      E_STATION_CTRL.STATION_ENABLE:
        IF (_wEnable = _wEnableProcess)
        THEN
          InitSerialTargets();
          _eProcessState            := E_STATION_STATE.STATION_DETECT_MOVER;
        END_IF
    END_CASE
END_CASE
//-----------------------------------------------------------------------------
// E_STATION_STATE.STATION_DETECT_MOVER: wait for any XtsStation to 
//                                       have a mover ready to enter
//-----------------------------------------------------------------------------
CASE _eProcessState
OF
  E_STATION_STATE.STATION_DETECT_MOVER:
    CASE _eProcessCmd
    OF
      E_STATION_CTRL.STATION_DISABLE:
        _eProcessState              := E_STATION_STATE.STATION_INIT;

      E_STATION_CTRL.STATION_ENABLE:
        IF (_wEnter > 0)            // at least one mover is asking for entry
        THEN
          _eDistributorTarget       := E_PROGRESS.PROGRESS_INVALID;

                                    // switch process state in order to tell process control
          _eProcessState            := E_STATION_STATE.STATION_MOVER_ENTER;
        END_IF
    END_CASE
END_CASE
//-----------------------------------------------------------------------------
//  E_STATION_STATE.STATION_MOVER_ENTER: check if infeed conditions are met, 
//                                       depending on type of process
//                                       Cmd from input (flow control)
//-----------------------------------------------------------------------------
CASE _eProcessState
OF
  E_STATION_STATE.STATION_MOVER_ENTER:
    CASE _eProcessCmd               // check input property
    OF
      E_STATION_CTRL.STATION_DISABLE:
        _eProcessState              := E_STATION_STATE.STATION_INIT;

      E_STATION_CTRL.STATION_MOVER_ENTER:
        FOR _nStn := _nLastStation TO _nFirstStation BY(-1) 
        DO
          CASE _stState^[_nStn].eState
          OF
          E_STATION_STATE.STATION_MOVER_ENTER,
          E_STATION_STATE.STATION_MOVER_IN_TARGET,
          E_STATION_STATE.STATION_PROCESS_START:
            IF GetBitDWord(_wEnter, (_nStn - _nFirstStation))
            THEN
              _stCtrl^[_nStn].eCmd  := E_STATION_CTRL.STATION_MOVER_ENTER;
            END_IF
          END_CASE
        END_FOR

        CASE _eType
        OF
          E_PROCESS_TYPE.PARALLEL_STRICT:
            IF (_wStart = _wEnable) // all who are enabled must have mover, in order to continue
            THEN
              _eProcessState        := E_STATION_STATE.STATION_PROCESS_START;
            END_IF

          E_PROCESS_TYPE.PARALLEL: 
            IF (_wStart = _wEnter)
            THEN
              _eProcessState        := E_STATION_STATE.STATION_PROCESS_START;
            END_IF

          E_PROCESS_TYPE.SERIAL:    // all who have work to do must have mover, in order to continue
            IF (_wMoverInStation > 0)
            THEN
              IF (_wStart = _wMoverInStation)
              THEN
                _eProcessState      := E_STATION_STATE.STATION_PROCESS_START;
              END_IF
            END_IF
        ELSE
          _eProcessState            := E_STATION_STATE.STATION_PROCESS_START;
        END_CASE

      E_STATION_CTRL.STATION_MOVER_SEND:  // flow control decided to skip process
        FOR _nStn := _nLastStation TO _nFirstStation BY(-1) 
        DO
          IF _bEnabledStation^[_nStn] AND 
             GetBitDWord(_wQueue, (_nStn-_nFirstStation))
          THEN
            IF (_TargetMask > 0)
            THEN
              // station is enabled AND has a mover in Queue to send
              _stCtrl^[_nStn].eCmd    := E_STATION_CTRL.STATION_MOVER_SEND;
            END_IF
          END_IF
        END_FOR
        IF (_wLeave > 0)            // wait for XtsStation to switch to outfeed
        THEN
          IF (_TargetMask > 0)
          THEN
            _eDistributorTarget       := DistributorTarget(_TargetMask);         // prepare target for mover
            IF (_eDistributorTarget = E_PROGRESS.PROGRESS_DONE)
            THEN
              _wStart                 := _wLeave;
              _eProcessState          := E_STATION_STATE.STATION_CHECK;
            END_IF
          END_IF
        END_IF 
    END_CASE
END_CASE
//-----------------------------------------------------------------------------
// synced process handshake on all stations in process
//-----------------------------------------------------------------------------
CASE _eProcessState                 // check output property
OF
  E_STATION_STATE.STATION_PROCESS_START:
    CASE _eType                     // decision for synced start varies for e_process_type
    OF
      E_PROCESS_TYPE.SERIAL:        // serial process must have had a mover waiting, which is now processed
      CASE _eProcessCmd             // check command input property
      OF
        E_STATION_CTRL.STATION_PROCESS_START,
        E_STATION_CTRL.STATION_PROCESS_DONE:
            IF (_wStart = _wMoverInStation)
            THEN
              _eProcessState          := E_STATION_STATE.STATION_PROCESS_DONE;
              FOR _nStn := _nLastStation TO _nFirstStation BY(-1) 
              DO
                // check for correct state on XtsStation
                CASE _stState^[_nStn].eState
                OF
                E_STATION_STATE.STATION_PROCESS_START:
                  _stCtrl^[_nStn].eCmd  := _eProcessCmd;
                END_CASE
              END_FOR
            END_IF
      END_CASE
    ELSE
      CASE _eProcessCmd             // check command input property
      OF
        E_STATION_CTRL.STATION_PROCESS_START,
        E_STATION_CTRL.STATION_PROCESS_DONE:
          IF (_wStart = _wEnter)
          THEN
            _eProcessState          := E_STATION_STATE.STATION_PROCESS_DONE;
            FOR _nStn := _nLastStation TO _nFirstStation BY(-1) 
            DO
              // check for correct state on XtsStation
              CASE _stState^[_nStn].eState
              OF
              E_STATION_STATE.STATION_PROCESS_START:
                _stCtrl^[_nStn].eCmd  := _eProcessCmd;
              END_CASE
            END_FOR
          END_IF
      END_CASE
    END_CASE
END_CASE
//-----------------------------------------------------------------------------
// synced process handshake on all stations in process
//-----------------------------------------------------------------------------
CASE _eProcessState                 // check output property
OF
  E_STATION_STATE.STATION_PROCESS_DONE:
    CASE _eProcessCmd               // check command input property
    OF
      E_STATION_CTRL.STATION_PROCESS_DONE: 
        FOR _nStn := _nLastStation TO _nFirstStation BY(-1) 
        DO
          _stCtrl^[_nStn].eCmd      := E_STATION_CTRL.STATION_PROCESS_DONE;
        END_FOR
        IF (_wLeave > 0)            // _wLeave tells us that xts station has mover to send
        THEN
          CASE _eType
          OF
            E_PROCESS_TYPE.SERIAL:
              _eProcessState        := E_STATION_STATE.STATION_CHECK;
              IF (_stState^[_nLastStation].nMoverId > 0)
              THEN
                PrepareLastSerialTarget();     // target for last xts station in serial process
              END_IF
    
              FOR _nStn := (_nLastStation - 1) TO _nFirstStation BY(-1) 
              DO
                _stCtrl^[_nStn].nTargetStation    := TO_USINT(_nSerialTarget[_nStn]);
              END_FOR
          ELSE
              IF (_TargetMask > 0)
              THEN
                ParallelTargets(_TargetMask);
                _eProcessState      := E_STATION_STATE.STATION_CHECK;
              END_IF
          END_CASE
        END_IF
    END_CASE
END_CASE
//-----------------------------------------------------------------------------
//-----------------------------------------------------------------------------
CASE _eProcessState
OF
  E_STATION_STATE.STATION_CHECK:    // TODO: implement procedure for target plausibility
    IF (_wTargetId > 0)             // simple check any target before switching to outfeed
    THEN
       _eProcessState               := E_STATION_STATE.STATION_MOVER_OUT;
(*
    ELSE                            // in case of invalid target, wait here for retry
      CASE _eType                   // retry varies for e_process_type
      OF
        E_PROCESS_TYPE.DISTRIBUTOR:
          IF (_eProcessCmd = E_STATION_CTRL.STATION_ENABLE)
          THEN
            // only distributor can land here directly; retry mover infeed
            _eProcessState          := E_STATION_STATE.STATION_MOVER_ENTER;
          END_IF
      ELSE
          IF (_eProcessCmd = E_STATION_CTRL.STATION_PROCESS_START)
          THEN
            // all other e_process_type must go back to process handshake
            _eProcessState          := E_STATION_STATE.STATION_PROCESS_DONE;
          END_IF
      END_CASE
*)
    END_IF
END_CASE
//-----------------------------------------------------------------------------
//-----------------------------------------------------------------------------
CASE _eProcessState
OF
  E_STATION_STATE.STATION_MOVER_OUT:
    IF (_wLeave = 0)                // all movers are gone
    THEN
      _eProcessState                := E_STATION_STATE.STATION_MOVER_GONE;

    ELSIF (_wLeave = _wStart)       // wait for everybody to be ready for send out
    THEN
      IF (_eProcessCmd = E_STATION_CTRL.STATION_MOVER_OUT)
      THEN
        FOR _nStn := _nLastStation TO _nFirstStation BY(-1) 
        DO
          CASE _stState^[_nStn].eState  // double check valid xts station state
          OF
            E_STATION_STATE.STATION_MOVER_OUT:
              IF (_stCtrl^[_nStn].nTargetStation > 0) // double check ticket on ctrl struct
              THEN
                _stCtrl^[_nStn].eCmd  := E_STATION_CTRL.STATION_MOVER_OUT;
              END_IF
          END_CASE
        END_FOR
      END_IF
    END_IF
END_CASE
//-----------------------------------------------------------------------------
//-----------------------------------------------------------------------------
CASE _eProcessState
OF
  E_STATION_STATE.STATION_MOVER_GONE:   // station is empty, quit mover gone and go back to the beginning
    FOR _nStn := _nLastStation TO _nFirstStation BY(-1) 
    DO
      _stCtrl^[_nStn].nTargetStation := 0;
      _stCtrl^[_nStn].eCmd      := E_STATION_CTRL.STATION_MOVER_GONE;
    END_FOR
    _eProcessState              := E_STATION_STATE.STATION_INIT;
END_CASE
END_METHOD

METHOD PRIVATE CycleStation
VAR
  _k                  : UINT;
END_VAR
IF NOT Check() THEN RETURN; END_IF

_wError                                   :=
_wErrorFatal                              := 0;

FOR _nStation := _nLastStation TO _nFirstStation BY(-1) 
DO
  // copy bit for enable station from input word to global array in GVL_PROCESS,
  //  - other processes read enabled state on mover out (PrepareTarget)
  _bEnabledStation^[_nStation]            := GetBitDWord(_wEnableProcess, (_nStation-_nFirstStation));

  IF (_stCtrl^[_nStation].nTargetStation > 0)
  THEN
    _wTargetId                            := SetBitDWord(_wTargetId,  (_nStation-_nFirstStation));
  ELSE
    _wTargetId                            := DelBitDWord(_wTargetId,  (_nStation-_nFirstStation));
  END_IF

  IF (_stState^[_nStation].nMoverId > 0)
  THEN
    _wMoverInStation                      := SetBitDWord(_wMoverInStation,  (_nStation-_nFirstStation));
  ELSE
    _wMoverInStation                      := DelBitDWord(_wMoverInStation,  (_nStation-_nFirstStation));
  END_IF

  IF (_stState^[_nStation].nQueue > 0)
  THEN
    _wQueue                               := SetBitDWord(_wQueue,  (_nStation-_nFirstStation));
  ELSE
    _wQueue                               := DelBitDWord(_wQueue,  (_nStation-_nFirstStation));
  END_IF

  CASE _stCtrl^[_nStation].eCmd
  OF
    E_STATION_CTRL.STATION_INIT:
      _stCtrl^[_nStation].nTargetStation  := 0;
      _wEnable                            := DelBitDWord(_wEnable, (_nStation-_nFirstStation));
      _wEnter                             := DelBitDWord(_wEnter,  (_nStation-_nFirstStation));
      _wStart                             := DelBitDWord(_wStart,  (_nStation-_nFirstStation));
      _wLeave                             := DelBitDWord(_wLeave,  (_nStation-_nFirstStation));

    E_STATION_CTRL.STATION_ENABLE:
      _wEnable                            := SetBitDWord(_wEnable, (_nStation-_nFirstStation));
  END_CASE

  CASE _stState^[_nStation].eState
  OF
    E_STATION_STATE.STATION_DISABLE:
      _wEnter                             := DelBitDWord(_wEnter,  (_nStation-_nFirstStation));

    E_STATION_STATE.STATION_MOVER_ENTER,
    E_STATION_STATE.STATION_MOVER_IN_TARGET:
      _wEnter                             := SetBitDWord(_wEnter,  (_nStation-_nFirstStation));
  
    E_STATION_STATE.STATION_PROCESS_START,
    E_STATION_STATE.STATION_PROCESS_DONE:
      _wStart                             := SetBitDWord(_wStart,  (_nStation-_nFirstStation));
  
    E_STATION_STATE.STATION_MOVER_OUT:
      _wLeave                             := SetBitDWord(_wLeave,  (_nStation-_nFirstStation));


    E_STATION_STATE.STATION_MOVER_GONE:
      _stCtrl^[_nStation].nTargetStation  := 0;
      _wStart                             := DelBitDWord(_wStart,  (_nStation-_nFirstStation));
      _wLeave                             := DelBitDWord(_wLeave,  (_nStation-_nFirstStation));
      _wEnable                            := DelBitDWord(_wEnable, (_nStation-_nFirstStation));
      _wEnter                             := DelBitDWord(_wEnter,  (_nStation-_nFirstStation));


    E_STATION_STATE.STATION_ERROR_LIST_STATION_ID_WRONG,  // wrong station ID in mover ticket (nTargetId written by preceeding station/process)
    E_STATION_STATE.STATION_ERROR_OUTFEED_TARGET_INVALID, // write correct target on station Ctrl.nTargetStation
    E_STATION_STATE.STATION_ERROR_INFEED_ERROR,           // clear mover error via Ctrl/State interface and retry on XTS station directly
    E_STATION_STATE.STATION_ERROR_OUTFEED_ERROR:          // clear mover error via Ctrl/State interface and retry on XTS station directly
      _wError                             := SetBitDWord(_wError,      (_nStation-_nFirstStation));

    E_STATION_STATE.STATION_ERROR_FATAL:
      _wErrorFatal                        := SetBitDWord(_wErrorFatal, (_nStation-_nFirstStation));

  END_CASE
END_FOR


_nProcessPerMinute          := 0;
// get mover counter
FOR _k := _nLastStation TO _nFirstStation BY(-1) 
DO
  _rtrigProcess[_k](
                  CLK       := (_stCtrl^[_k].eCmd = E_STATION_CTRL.STATION_MOVER_OUT));

  IF _rtrigProcess[_k].Q
  THEN
    _nMoverCount[_k]        := _nMoverCount[_k] + 1;
  END_IF
  
  IF _tonPartsperMinute.Q
  THEN
    _nMoverPerMinute^[_k]   := _nMoverCount[_k] - _nMoverCountOld[_k];
    _nMoverCountOld  [_k]   := _nMoverCount[_k];
  END_IF
  _nProcessPerMinute        := _nProcessPerMinute + _nMoverPerMinute^[_k]; 
END_FOR

IF _tonPartsperMinute.q
THEN
  _tonPartsperMinute(
                  IN        :=FALSE);
END_IF

_tonPartsperMinute(
                  IN        := TRUE, 
                  PT        := T#60S);
END_METHOD

METHOD PUBLIC DelBitDWord : DWORD
VAR_INPUT
  inVal   : DWORD;
  bitNo   : DWORD;
END_VAR
VAR
  wConst : DWORD := 1;
END_VAR
IF ( inVal AND SHL( wConst,bitNo MOD 16 ) ) > 0 THEN
  DelBitDWord := inVal XOR (SHL( wConst,bitNo MOD 16 ));
ELSE
  DelBitDWord := inVal;
END_IF
END_METHOD

METHOD DistributorTarget : e_progress
VAR_INPUT
  wTarget         : DWORD; // bits for target stations to be used
END_VAR
VAR_INST
  _eResult        : E_PROGRESS;
  {attribute 'displaymode':='bin'}
  _wtg            : DWORD;
END_VAR
IF NOT Check() THEN RETURN; END_IF
_wtg := wTarget;

// check if target station is enabled
IF GetBitDWord(wTarget, (_nTarget))
THEN
  _nPreparedTarget[_stState^[_nFirstStation].nMoverId]  := _nLastTarget - _nTarget;
  _stCtrl^[_nFirstStation].nTargetStation               := TO_USINT(_nLastTarget - _nTarget);
  _eResult                                              := E_PROGRESS.PROGRESS_DONE;
ELSE
  _eResult                                              := e_progress.PROGRESS_BUSY;
END_IF

_nTarget                      := _nTarget + 1;
IF (_nLastTarget - _nTarget < _nFirstTarget)
THEN
  _nTarget                    := 0;
END_IF

DistributorTarget                                       := _eResult;
END_METHOD

PROPERTY EnabledStation : POINTER TO ARRAY[1..XTS_Parameter.MAX_STATION]  OF bool;
SET
_bEnabledStation := EnabledStation;
END_SET
END_PROPERTY

PROPERTY EnableProcess : dword
GET
EnableProcess := _wEnableProcess;
END_GET
SET
_wEnableProcess := EnableProcess;
END_SET
END_PROPERTY

METHOD PUBLIC GetBitDWord : BOOL
VAR_INPUT
  inVal   : DWORD;
  bitNo   : DINT;
END_VAR
VAR
  wConst : DWORD := 1;
END_VAR
IF ( inVal AND SHL( wConst,DINT_TO_SINT(bitNo) MOD 32 ) ) > 0
THEN
  GetBitDWord := TRUE;
ELSE
  GetBitDWord := FALSE;
END_IF
END_METHOD

METHOD PUBLIC Init : BOOL
VAR
  _nStn     : UINT;
END_VAR
IF NOT (_nLastStation   > 0) OR
   NOT (_nFirstStation  > 0) OR
   NOT (_nLastStation   < MAX_STATION+1) OR
   NOT (_nFirstStation  < MAX_STATION+1)
THEN
  Init := FALSE;
  _eProcessState                := E_STATION_STATE.STATION_NO_INIT;
ELSE
  _eProcessState                := E_STATION_STATE.STATION_NO_INIT;

  FOR _nStn := _nLastStation TO _nFirstStation BY(-1) 
  DO
    _stCtrl^[_nStn].eCmd        := E_STATION_CTRL.STATION_INIT;
    _stCtrl^[_nStn].nMask       := 0;

    IF NOT (_stState^[_nStn].eState = E_STATION_STATE.STATION_INIT)
    THEN
      Init := FALSE;
      RETURN;
    END_IF  
  END_FOR

  memset(ADR(_nMoverCount),       0, SIZEOF(_nMoverCount));
  memset(ADR(_nMoverCountOld),    0, SIZEOF(_nMoverCountOld));
  _nTarget                      := 0;

  _eProcessState                := E_STATION_STATE.STATION_INIT;

  Init := TRUE;
END_IF
END_METHOD

METHOD PRIVATE InitSerialTargets
VAR
  _k    : uint;
END_VAR

IF NOT (_nStationCount > 1)
THEN
  RETURN;
END_IF

// serial process must always have at least two xts stations to work with
FOR _nStation := _nLastStation TO _nFirstStation+1 BY(-1) 
DO
  IF (_bEnabledStation^[_nStation])
  THEN
    _nSerialTarget[_nStation-1] := _nStation;
  END_IF
END_FOR
END_METHOD

PROPERTY MoverCountInQueue : uint
GET
VAR
  _nTmp   : UINT;
  _nCount : uint;
END_VAR
IF NOT (_nStationCount > 0)
THEN
  MoverCountInQueue := 0;
  RETURN;
END_IF

FOR _nTmp := _nLastStation TO _nFirstStation BY(-1)
DO
  _nCount := _nCount + _stState^[_nTmp].nQueue;
END_FOR

MoverCountInQueue := _nCount;
END_GET
END_PROPERTY

PROPERTY MoverInQueue : Bool
GET
MoverInQueue  := SEL((_wQueue > 0), FALSE, TRUE);
END_GET
END_PROPERTY

PROPERTY MoverPerMinute : pointer to ARRAY[1..XTS_Parameter.MAX_STATION]  OF UINT
SET
_nMoverPerMinute  := MoverPerMinute;
END_SET
END_PROPERTY

METHOD PRIVATE ParallelTargets : E_PROGRESS
VAR_INPUT
  wTarget         : DWORD; // bits for target stations to be used
END_VAR
VAR_INST
  {attribute 'displaymode':='bin'}
  _wtg            : DWORD;
  _nt,
  _idxStation     : UINT;
END_VAR
IF NOT Check() THEN RETURN; END_IF
_wtg := wTarget;


FOR _idxStation := _nLastStation TO _nFirstStation BY(-1) 
DO
  _nt                           := _nLastTarget - _nTarget;

  // check if target station is enabled
  IF GetBitDWord(wTarget, (_nTarget))
  THEN
    IF (_stState^[_idxStation].nMoverId <> 0)
    THEN
      _nPreparedTarget[_stState^[_idxStation].nMoverId]  := _nt;
      _stCtrl^[_idxStation].nTargetStation               := TO_USINT(_nt);
    END_IF
  END_IF

  _nTarget                      := _nTarget + 1;
  IF (_nLastTarget - _nTarget < _nFirstTarget)
  THEN
    _nTarget                    := 0;
  END_IF
END_FOR
END_METHOD

METHOD PRIVATE PrepareLastSerialTarget
VAR
  _nt   : uint;
END_VAR

_nt                           := _nLastTarget - _nTarget;
_nTarget                      := _nTarget + 1;

// check if target station is enabled
IF (_bEnabledStation^[_nt])
THEN
  _nPreparedTarget[_stState^[_nLastStation].nMoverId]  := _nt;
  _stCtrl^[_nLastStation].nTargetStation               := TO_USINT(_nt);
END_IF

IF (_nLastTarget - _nTarget < _nFirstTarget)
THEN
  _nTarget                    := 0;
END_IF
END_METHOD

PROPERTY ProcessCmd : E_STATION_CTRL
SET
_eProcessCmd := ProcessCmd;
END_SET
END_PROPERTY

PROPERTY ProcessPerMinute : uint
GET
ProcessPerMinute := _nProcessPerMinute;
END_GET
END_PROPERTY

PROPERTY ProcessState : E_STATION_STATE
GET
ProcessState := _eProcessState;
END_GET
END_PROPERTY

PROPERTY ProcessType : e_process_type
GET
ProcessType := _eType;
END_GET
SET
_eType := ProcessType;
END_SET
END_PROPERTY

METHOD PUBLIC SetBitDWord : DWORD
VAR_INPUT
  inVal   : DWORD;
  bitNo   : DWORD;
END_VAR
VAR
  wConst  : DWORD := 1;
END_VAR
SetBitDWord := inVal OR SHL( wConst,bitNo MOD 32 );
END_METHOD

METHOD PUBLIC SetBitWord : WORD
VAR_INPUT
  inVal   : WORD;
  bitNo   : DINT;
END_VAR
VAR
  wConst  : WORD := 1;
END_VAR
SetBitWord := inVal OR SHL( wConst,bitNo MOD 16 );
END_METHOD

PROPERTY StationCount : uint
GET
StationCount := _nStationCount;
END_GET
END_PROPERTY

PROPERTY StationCtrl : pointer to ARRAY[1..XTS_Parameter.MAX_STATION]  OF ST_STATION_CTRL;
SET
_stCtrl := StationCtrl;
END_SET
END_PROPERTY

PROPERTY StationFirst : uint
GET
StationFirst := _nFirstStation;
END_GET
SET
_nFirstStation := StationFirst;
END_SET
END_PROPERTY

PROPERTY StationLast : uint
GET
StationLast := _nLastStation;
END_GET
SET
_nLastStation := StationLast;
END_SET
END_PROPERTY

PROPERTY StationState : POINTER TO ARRAY[1..XTS_Parameter.MAX_STATION]  OF ST_STATION_STATE
SET
_stState := StationState;
END_SET
END_PROPERTY

PROPERTY TargetFirst : uint
GET
TargetFirst := _nFirstTarget;
END_GET
SET
_nFirstTarget := TargetFirst;
END_SET
END_PROPERTY

PROPERTY TargetLast : uint
GET
TargetLast := _nLastTarget;
END_GET
SET
_nLastTarget := TargetLast;
END_SET
END_PROPERTY

PROPERTY TargetMask : dword
GET
TargetMask := _TargetMask;
END_GET
SET
_TargetMask := TargetMask;
END_SET
END_PROPERTY

END_FUNCTION_BLOCK

// ---- XTS/XtsStation/fb_Station.TcPOU
//---------------------------------------------------------------------------------------------------------------
//
//  HAUD 2023.03.07
//
//  - XTS_TRANSPORT_LAYER
//
//  fb_Station
//  - handshake with extern control for mover transport through station
//
//---------------------------------------------------------------------------------------------------------------
// This SOFTWARE is provided as an Exemple by THE PROVIDER "as is" and "with all faults." THE PROVIDER makes no 
// representations or warranties of any kind concerning the safety, suitability, lack of viruses, inaccuracies, 
// typographical errors, or other harmful components of this SOFTWARE. There are inherent dangers in the use of 
// any software, and you are solely responsible for determining whether this SOFTWARE is compatible with your 
// equipment and other software installed on your equipment. You are also solely responsible for the protection 
// of your equipment and backup of your data, and THE PROVIDER will not be liable for any damages you may suffer 
// in connection with using, modifying, or distributing this SOFTWARE.
//---------------------------------------------------------------------------------------------------------------
FUNCTION_BLOCK fb_Station IMPLEMENTS I_XtsTransport_Station
VAR
  _nStationId                 : UINT;         // why is Gamora?

  _sState                     : STRING(255);  // additional output for Check()

  _eInitList                  : E_PROGRESS;   // linked list initialization progress

  _eFatalError                : E_STATION_STATE;

  // pointer to all stations
  _stCtrl                     : REFERENCE TO ARRAY[1..MAX_STATION]  OF ST_STATION_CTRL;
  _stState                    : REFERENCE TO ARRAY[1..MAX_STATION]  OF ST_STATION_STATE;

  // local copy of me
  _stStationCtrl              : ST_STATION_CTRL;
  _stStationState             : ST_STATION_STATE;

  _ItfStation                 : REFERENCE TO ARRAY[1..MAX_STATION]  OF I_Station_LinkedList;  // access to all stations lists
  _ItfMover                   : REFERENCE TO ARRAY[1..MAX_MOVER]    OF I_XtsTransport_Mover;  // access to mover methods

  // station related data
  _rMoverOffset               : REFERENCE TO ARRAY[1..MAX_STATION]  OF T_NEST_OFFSET;         // static offsets for station
  _stParameter                : REFERENCE TO ARRAY[1..MAX_STATION]  OF ST_STATION_PARAMETER;  // station parameter (where, how fast, how many stops)

  // mover axis ref for info
  _Mover                      : REFERENCE TO ARRAY[1..MAX_MOVER]    OF AXIS_REF;              // read from AXIS_REF

  // linked list result struct
  _stListEnter,
  _stListTarget,
  _stListDelete               : ST_STATION_LIST_RESULT;   // struct with result and ticket data

  _stMoverDataSend,
  _stMoverData                : ST_STATION_MOVER_DATA;    // mover ticket data

  _stInfeed,
  _stOutfeed                  : ST_MOVE_DATA;             // position and dynamic constraints of movement

  // work vars
  _Result                     : E_PROGRESS;
  _eState                     : E_PROGRESS;

  _nNest,
  _nMoverDetected,
  _nMoverInStation,
  _nTargetStation,
  _ix                         : UINT;

  _rModActPosFetch            : LREAL;
  _stMsg                      : ST_Message;
  _eMessageLevel              : E_MessageType;
END_VAR

METHOD PRIVATE Check : BOOL
VAR_INPUT
END_VAR
IF NOT (_nStationId > 0) OR
       (_nStationId > MAX_STATION)
THEN
  _sState                     := 'invalid nStationId';
  RETURN;
END_IF

IF NOT __ISVALIDREF(_stCtrl)
THEN
  _sState                     := '_stCtrl: missing pointer';
  RETURN;
END_IF

IF NOT __ISVALIDREF(_stState)
THEN
  _sState                     := '_stState: missing pointer';
  RETURN;
END_IF

IF NOT __ISVALIDREF(_ItfStation)
THEN
  _sState                     := '_ItfStation: missing interface';
  RETURN;
END_IF

IF NOT __ISVALIDREF(_ItfMover)
THEN
  _sState                     := '_ItfMover: missing interface';
  RETURN;
END_IF

IF NOT __ISVALIDREF(_rMoverOffset)
THEN
  _sState                     := '_rMoverOffset: missing pointer';
  RETURN;
END_IF

IF NOT __ISVALIDREF(_stParameter)
THEN
  _sState                     := '_stParameter: missing pointer';
  RETURN;
END_IF

IF NOT __ISVALIDREF(_Mover)
THEN
  _sState                     := '_Mover: missing pointer';
  RETURN;
END_IF


_sState                       := 'CHECK_DONE';
Check                         := TRUE;
END_METHOD

PROPERTY Ctrl : reference to ARRAY[1..MAX_STATION] OF ST_STATION_CTRL
SET
_stCtrl ref= Ctrl;
END_SET
END_PROPERTY

METHOD Cycle
// check pointer and interface
IF NOT Check() THEN RETURN; END_IF

_stMsg.eDevice                        := e_Device.XtsStation + _nStationId;

IF (_stCtrl[_nStationId].eCmd <> _stStationCtrl.eCmd)
THEN
  _stMsg.eType                        := E_MessageType.eMessageVerbose;
  _stMsg.eSubdevice                   := StationControl;
  _stMsg.iErrorNumber                 := 0;
  _stMsg.sText                        := TO_STRING(_stCtrl[_nStationId].eCmd);
  IF (_eMessageLevel = E_MessageType.eMessageVerbose)
  THEN
    f_MessageSet(_stMsg);
  END_IF
END_IF

//-----------------------------------------------------------------------------
// copy ctrl to local
//-----------------------------------------------------------------------------
_stStationCtrl                        := _stCtrl[_nStationId];


// direct from interface
CASE _stCtrl[_nStationId].eCmd
OF
  E_STATION_CTRL.STATION_INIT:        // commanded init from cyclic interface
    _eInitList                        := Init();
    RETURN;
END_CASE

//-----------------------------------------------------------------------------
//-----------------------------------------------------------------------------
CASE _stStationState.eState
OF
  E_STATION_STATE.STATION_NO_INIT:    // startup state in first PLC cycle, init linked list required
    _eInitList                        := Init();

  E_STATION_STATE.STATION_INIT:       // switch state as reserve for anything you might add here
    _stStationState.nMoverId          := 0;
    _stStationState.eState            := E_STATION_STATE.STATION_DISABLE;
END_CASE
//-----------------------------------------------------------------------------
//-----------------------------------------------------------------------------
CASE _stStationState.eState
OF
  E_STATION_STATE.STATION_DISABLE:    // end state after first PLC cycle startup; wait state after commanded disable
    IF (_stStationCtrl.eCmd = E_STATION_CTRL.STATION_ENABLE)
    THEN
      _stStationState.eState          := E_STATION_STATE.STATION_ENABLE;
    END_IF


  E_STATION_STATE.STATION_ENABLE:     // double check commanded enable and clear work vars
    IF (_stStationCtrl.eCmd = E_STATION_CTRL.STATION_ENABLE)
    THEN
      memset(ADR(_stListEnter),    0, SIZEOF(_stListEnter));

      _eState                         := E_PROGRESS.PROGRESS_INIT;  // work var for nested case
      _stStationState.eState          := E_STATION_STATE.STATION_DETECT_MOVER;

      _stMsg.eType                    := E_MessageType.eMessageVerbose;
      IF (_eMessageLevel = E_MessageType.eMessageVerbose)
      THEN
        LogState(_stMsg.eType);
      END_IF
    END_IF
END_CASE
//-----------------------------------------------------------------------------
//-----------------------------------------------------------------------------
CASE _stStationState.eState
OF
  E_STATION_STATE.STATION_DETECT_MOVER:// wait state for mover detection
    CASE _eState
    OF
      E_PROGRESS.PROGRESS_INIT:
        IF (_stStationCtrl.eCmd = E_STATION_CTRL.STATION_DISABLE) // check for commanded disable
        THEN
          IF (_eMessageLevel = E_MessageType.eMessageVerbose)
          THEN
            _stMsg.eType              := E_MessageType.eMessageVerbose;
            _stMsg.eSubdevice         := Stationstate;
            _stMsg.iErrorNumber       := _stStationState.nMoverId;
            _stMsg.sText              := concat(TO_STRING(_stStationState.eState), ': ');
            _stMsg.sText              := concat(_stMsg.sText, TO_STRING(E_STATION_STATE.STATION_DISABLE));
            f_MessageSet(_stMsg);
          END_IF
          _stStationState.eState      := E_STATION_STATE.STATION_DISABLE; // go back and wait, no matter the queue

        ELSIF (_ItfStation[_nStationId].Count > 0)
        THEN
          // someone entered something in my list
          _stListEnter                := _ItfStation[_nStationId].GetHead();
          _eState                     := E_PROGRESS.PROGRESS_BUSY;

          IF (_eMessageLevel = E_MessageType.eMessageVerbose)
          THEN
            _stMsg.eType              := E_MessageType.eMessageVerbose;
            _stMsg.eSubdevice         := Stationstate;
            _stMsg.iErrorNumber       := _stStationState.nMoverId;
            _stMsg.sText              := concat(TO_STRING(_stStationState.eState), ': ');
            _stMsg.sText              := concat(_stMsg.sText, TO_STRING(_eState));
            f_MessageSet(_stMsg);
          END_IF
        END_IF
    END_CASE
    CASE _eState
    OF
      E_PROGRESS.PROGRESS_BUSY:
        IF (_stListEnter.wState = 0)  // GetHead() without error
        THEN
          _stMsg.eType                := E_MessageType.eMessageVerbose;
          _stMsg.eSubdevice           := e_Subdevice.StationGetHead;
          _stMsg.iErrorNumber         := _stListEnter.stData.nMoverId;
          _stMsg.sText                := '';
          IF (_eMessageLevel = E_MessageType.eMessageVerbose)
          THEN
            f_MessageSet(_stMsg);
          END_IF

          // list is giving head as result
          _stMoverData                := _stListEnter.stData; // copy ticket from list result
          _eState                     := E_PROGRESS.PROGRESS_PREPARE;

          IF (_eMessageLevel = E_MessageType.eMessageVerbose)
          THEN
            _stMsg.eType              := E_MessageType.eMessageVerbose;
            _stMsg.eSubdevice         := Stationstate;
            _stMsg.iErrorNumber       := _stStationState.nMoverId;
            _stMsg.sText              := concat(TO_STRING(_stStationState.eState), ': ');
            _stMsg.sText              := concat(_stMsg.sText, TO_STRING(_eState));
            f_MessageSet(_stMsg);
          END_IF
        ELSE
          // the thing that must not be: GetHead() with error
          _stStationState.eState      := E_STATION_STATE.STATION_ERROR_LIST_GET_HEAD_FAULT;

          _stMsg.eType                := E_MessageType.eMessageError;
          LogState(_stMsg.eType);
        END_IF
    END_CASE
    CASE _eState
    OF
      E_PROGRESS.PROGRESS_PREPARE:    // check ticket (list entry)
        // check target assignement
        IF NOT (_stMoverData.nTargetStation = _nStationId)
        THEN
          // for whom the mover calls
          // wrong address, right mover?
          _stStationState.eState      := E_STATION_STATE.STATION_ERROR_LIST_STATION_ID_WRONG;

          _stMsg.eType                := E_MessageType.eMessageWarning;
          LogState(_stMsg.eType);
        ELSE
          // it's a me
          _nMoverDetected             := _stMoverData.nMoverId;

          IF (_nMoverDetected < 1) OR
             (_nMoverDetected > MAX_MOVER)
          THEN
            // out of range the mover must not be
            _stStationState.eState    := E_STATION_STATE.STATION_ERROR_LIST_MOVER_ID_INVALID;

            _stMsg.eType              := E_MessageType.eMessageError;
            LogState(_stMsg.eType);
          ELSE
            memset(ADR(_stListDelete),   0, SIZEOF(_stListDelete)); // clear work var
            _eState                   := E_PROGRESS.PROGRESS_INIT;

            // prepare station state for new mover
            _stStationState.nMoverId  := TO_USINT(_nMoverDetected); // who has arrived
            _stStationState.nMask     := _stMoverData.nMask;        // how many stops have to be made
            _stStationState.eState    := E_STATION_STATE.STATION_MOVER_ENTER; // go ask for permission to enter

            IF (_eMessageLevel = E_MessageType.eMessageVerbose)
            THEN
              _stMsg.eType            := E_MessageType.eMessageVerbose;
              _stMsg.eSubdevice       := Stationstate;
              _stMsg.iErrorNumber     := _stStationState.nMoverId;
              _stMsg.sText            := concat(TO_STRING(_stStationState.eState), ': ');
              _stMsg.sText            := concat(_stMsg.sText, TO_STRING(_eState));
              f_MessageSet(_stMsg);
            END_IF
          END_IF
        END_IF
    END_CASE
END_CASE
//-----------------------------------------------------------------------------
//-----------------------------------------------------------------------------
CASE _stStationState.eState
OF
  E_STATION_STATE.STATION_MOVER_ENTER:          // requesting permission for mover to enter station
    CASE _eState
    OF
      E_PROGRESS.PROGRESS_INIT:

        CASE _stStationCtrl.eCmd
        OF
          E_STATION_CTRL.STATION_DISABLE:       // control decided to disable, mover will wait
            _stStationState.eState    := E_STATION_STATE.STATION_DISABLE;

            IF (_eMessageLevel = E_MessageType.eMessageVerbose)
            THEN
              _stMsg.eType            := E_MessageType.eMessageVerbose;
              LogState(_stMsg.eType);
            END_IF

          E_STATION_CTRL.STATION_MOVER_ENTER:   // control decided to let mover enter
            _nNest                    := 1;     // default nest/StopPos
            _eState                   := E_PROGRESS.PROGRESS_BUSY;

            IF (_eMessageLevel = E_MessageType.eMessageVerbose)
            THEN
              _stMsg.eType            := E_MessageType.eMessageVerbose;
              _stMsg.eSubdevice         := Stationstate;
              _stMsg.iErrorNumber       := _stStationState.nMoverId;
              _stMsg.sText              := concat(TO_STRING(_stStationState.eState), ': ');
              _stMsg.sText              := concat(_stMsg.sText, TO_STRING(_eState));
              f_MessageSet(_stMsg);
            END_IF

            FOR _ix := 1 TO _stParameter[_nStationId].nConfiguredStopCount
            DO
              IF GetBitWord(_stMoverData.nMask, _ix-1)
              THEN
                _nNest                := _ix;
                EXIT;
              END_IF
            END_FOR

          E_STATION_CTRL.STATION_MOVER_SEND:    // control decided to send mover away
            _stOutfeed.rDistance      := 0.5 * _stParameter[_nStationId].rReleaseDistance;
            _stStationState.eState    := E_STATION_STATE.STATION_MOVER_OUT;

            IF (_eMessageLevel = E_MessageType.eMessageVerbose)
            THEN
              _stMsg.eType            := E_MessageType.eMessageVerbose;
              LogState(_stMsg.eType);
            END_IF
        END_CASE
    END_CASE
    CASE _eState
    OF
      E_PROGRESS.PROGRESS_BUSY:
        MoveData();

        // check if infeed movement has to cross modulo turn
        _rModActPosFetch              := _Mover[_stMoverData.nMoverId].NcToPlc.ModuloActPos;

        IF (_rModActPosFetch > _stInfeed.rPos + _stParameter[_nStationId].rReleaseDistance)
        THEN
          _stInfeed.rPos            := _stInfeed.rPos + TO_REAL(_ItfMover[_stMoverData.nMoverId].RailLength);
        END_IF

        _stStationState.eState        := E_STATION_STATE.STATION_MOVER_IN_TARGET;

        IF (_eMessageLevel = E_MessageType.eMessageVerbose)
        THEN
          _stMsg.eType                := E_MessageType.eMessageVerbose;
          LogState(_stMsg.eType);
        END_IF
    END_CASE
END_CASE
//-----------------------------------------------------------------------------
//-----------------------------------------------------------------------------
CASE _stStationState.eState
OF
  E_STATION_STATE.STATION_MOVER_IN_TARGET:
    _Result := _ItfMover[_stMoverData.nMoverId].MoveToPosCa(TRUE, _stInfeed);

    IF (_Result = E_PROGRESS.PROGRESS_DONE)
    THEN
      // mother! has arrived
      _ItfMover[_stMoverData.nMoverId].MoveToPosCa(FALSE, _stInfeed);
      _stStationState.eState          := E_STATION_STATE.STATION_PROCESS_START;

      IF (_eMessageLevel = E_MessageType.eMessageVerbose)
      THEN
        _stMsg.eType                  := E_MessageType.eMessageVerbose;
        LogState(_stMsg.eType);
      END_IF
    ELSE
      IF (_Result = E_PROGRESS.PROGRESS_ERROR)
      THEN
        _ItfMover[_stMoverData.nMoverId].MoveToPosCa(FALSE, _stInfeed);
        _stStationState.eState        := E_STATION_STATE.STATION_ERROR_INFEED_ERROR;

        _stMsg.eType                  := E_MessageType.eMessageError;
        LogState(_stMsg.eType);
      END_IF 
    END_IF
END_CASE
//-----------------------------------------------------------------------------
//-----------------------------------------------------------------------------
CASE _stStationState.eState
OF
  E_STATION_STATE.STATION_PROCESS_START:
    IF (_stStationCtrl.eCmd = E_STATION_CTRL.STATION_PROCESS_START) OR  // double handshake, your choice
       (_stStationCtrl.eCmd = E_STATION_CTRL.STATION_PROCESS_DONE)      // single handshake, your choice
    THEN
      // clear bit in mask when started/done
      _stStationState.nMask           := TO_USINT(DelBitWord(TO_WORD(_stStationState.nMask), _nNest-1));
      _stStationState.eState          := E_STATION_STATE.STATION_PROCESS_DONE;

      IF (_eMessageLevel = E_MessageType.eMessageVerbose)
      THEN
        _stMsg.eType                  := E_MessageType.eMessageVerbose;
        LogState(_stMsg.eType);
      END_IF
    END_IF
END_CASE
//-----------------------------------------------------------------------------
//-----------------------------------------------------------------------------
CASE _stStationState.eState
OF
  E_STATION_STATE.STATION_PROCESS_DONE:
    IF (_stStationCtrl.eCmd = E_STATION_CTRL.STATION_PROCESS_DONE)
    THEN
      _stStationState.eState          := E_STATION_STATE.STATION_CHECK;
    END_IF
END_CASE
//-----------------------------------------------------------------------------
//-----------------------------------------------------------------------------
CASE _stStationState.eState
OF
  E_STATION_STATE.STATION_CHECK:
    IF (_stStationState.nMask = 0)
    THEN
      // mover has to leave
      _stInfeed.rDistance           := _stParameter[_nStationId].rReleaseDistance;
      _stStationState.eState          := E_STATION_STATE.STATION_MOVER_OUT;

      IF (_eMessageLevel = E_MessageType.eMessageVerbose)
      THEN
        _stMsg.eType                  := E_MessageType.eMessageVerbose;
        LogState(_stMsg.eType);
      END_IF
    ELSE
      // _stStationState.nMask <> 0
      FOR _ix := 1 TO MAX_STATION_NEST
      DO
        IF NOT (_ix > _stParameter[_nStationId].nConfiguredStopCount)
        THEN
          IF GetBitWord(_stStationState.nMask, _ix-1)
          THEN
            // more work to do
            _stStationState.eState    := E_STATION_STATE.STATION_CHECK_NEST;
            _nNest                    := _ix;

            IF (_eMessageLevel = E_MessageType.eMessageVerbose)
            THEN
              _stMsg.eType            := E_MessageType.eMessageVerbose;
              LogState(_stMsg.eType);
            END_IF
            EXIT;
          END_IF
        ELSE
          IF GetBitWord(_stStationState.nMask, _ix-1)
          THEN
            // not configured, not worked
            _stMsg.eType              := E_MessageType.eMessageWarning;
            _stMsg.eSubdevice         := Stationstate;
            _stMsg.iErrorNumber       := _ix;
            _stMsg.sText              := concat(TO_STRING(_stStationState.eState), ': ');
            _stMsg.sText              := concat(_stMsg.sText, Tc2_Utilities.BYTE_TO_BINSTR(_stStationState.nMask, TO_INT(MAX_STATION_NEST)));
            f_MessageSet(_stMsg);

            _stStationState.nMask     := TO_USINT(DelBitWord(TO_WORD(_stStationState.nMask), _ix-1));
          END_IF
        END_IF
      END_FOR
    END_IF
END_CASE
//-----------------------------------------------------------------------------
//-----------------------------------------------------------------------------
CASE _stStationState.eState
OF
  E_STATION_STATE.STATION_CHECK_NEST:
    MoveData();

    IF (_stStationCtrl.eCmd = E_STATION_CTRL.STATION_MOVER_ENTER)
    THEN
      _stStationState.eState            := E_STATION_STATE.STATION_MOVER_IN_TARGET;
  
      IF (_eMessageLevel = E_MessageType.eMessageVerbose)
      THEN
        _stMsg.eType                    := E_MessageType.eMessageVerbose;
        LogState(_stMsg.eType);
      END_IF
    END_IF
END_CASE
//-----------------------------------------------------------------------------
//-----------------------------------------------------------------------------
CASE _stStationState.eState
OF
  E_STATION_STATE.STATION_MOVER_OUT:
    IF (_stStationCtrl.eCmd = E_STATION_CTRL.STATION_MOVER_OUT)
    THEN
      IF (_stStationCtrl.nTargetStation < 1) OR  
         (_stStationCtrl.nTargetStation > MAX_STATION)
      THEN
        _stStationState.eState        := E_STATION_STATE.STATION_ERROR_OUTFEED_TARGET_INVALID;

        _stMsg.eType                  := E_MessageType.eMessageError;
        LogState(_stMsg.eType);
      ELSE
        _stListDelete                 := _ItfStation[_nStationId].RemoveHeadValue();

        IF (_stListDelete.wState <> 0)
        THEN
          _stStationState.eState      := E_STATION_STATE.STATION_ERROR_LIST_REMOVE_HEAD_FAULT;

          _stMsg.eType                := E_MessageType.eMessageError;
          LogState(_stMsg.eType);

        ELSE
          _stMsg.eType                := E_MessageType.eMessageVerbose;
          _stMsg.eSubdevice           := e_Subdevice.StationRemoveHeadValue;
          _stMsg.iErrorNumber         := _stStationState.nMoverId;
          _stMsg.sText                := '';
          IF (_eMessageLevel = E_MessageType.eMessageVerbose)
          THEN
            f_MessageSet(_stMsg);
          END_IF

          memset(ADR(_stListTarget),   0, SIZEOF(_stListTarget));

          MoverOut();
          _stStationState.eState      := E_STATION_STATE.STATION_MOVER_RELEASE;

          IF (_eMessageLevel = E_MessageType.eMessageVerbose)
          THEN
            _stMsg.eType              := E_MessageType.eMessageVerbose;
            LogState(_stMsg.eType);
          END_IF
        END_IF
      END_IF
    END_IF
END_CASE
//-----------------------------------------------------------------------------
//-----------------------------------------------------------------------------
CASE _stStationState.eState
OF
  E_STATION_STATE.STATION_MOVER_RELEASE:
    _Result                           := _ItfMover[_stMoverDataSend.nMoverId].SendToModuloPosCa(TRUE, _stOutfeed);

    IF (_Result = E_PROGRESS.PROGRESS_DONE)
    THEN
      // add entry in target station list
      _stListTarget                   := _ItfStation[_stMoverDataSend.nTargetStation].AddTailValue(_stMoverDataSend);

      IF (_stListTarget.wState <> 0)
      THEN
        _stStationState.eState        := E_STATION_STATE.STATION_ERROR_LIST_ADD_TAIL_FAULT;
        _stMsg.eType                  := E_MessageType.eMessageError;
        LogState(_stMsg.eType);

      ELSE
        IF (_eMessageLevel = E_MessageType.eMessageVerbose)
        THEN
          _stMsg.eType                := E_MessageType.eMessageVerbose;
          _stMsg.eSubdevice           := e_Subdevice.StationAddTail;
          _stMsg.iErrorNumber         := _stStationState.nMoverId;
          _stMsg.sText                := concat('TargetStation: ', TO_STRING(_stListTarget.stData.nTargetStation));
          f_MessageSet(_stMsg);
        END_IF

        _stStationState.eState        := E_STATION_STATE.STATION_MOVER_GONE;

        IF (_eMessageLevel = E_MessageType.eMessageVerbose)
        THEN
          _stMsg.eType                := E_MessageType.eMessageVerbose;
          LogState(_stMsg.eType);
        END_IF
      END_IF
    ELSIF (_Result = E_PROGRESS.PROGRESS_ERROR)
    THEN
      _stStationState.eState          := E_STATION_STATE.STATION_ERROR_OUTFEED_ERROR;
      _stMsg.eType                    := E_MessageType.eMessageError;
      LogState(_stMsg.eType);
    END_IF
END_CASE
//-----------------------------------------------------------------------------
//-----------------------------------------------------------------------------
CASE _stStationState.eState
OF
  E_STATION_STATE.STATION_MOVER_GONE:
    _ItfMover[_stMoverDataSend.nMoverId].SendToModuloPosCa(FALSE, 
                                                      _stOutfeed);

    memset(ADR(_stMoverData),  0, SIZEOF(_stMoverData));

    _stStationState.nMask             := 0;
    _stStationState.nMoverId          := 0;

    IF (_stStationCtrl.eCmd = E_STATION_CTRL.STATION_MOVER_GONE)
    THEN
      _stStationState.eState          := E_STATION_STATE.STATION_INIT;

      IF (_eMessageLevel = E_MessageType.eMessageVerbose)
      THEN
        _stMsg.eType                  := E_MessageType.eMessageVerbose;
        LogState(_stMsg.eType);
      END_IF
    END_IF
END_CASE
//-----------------------------------------------------------------------------
//-----------------------------------------------------------------------------
_sState                               := TO_STRING(_stStationState.eState);
//-----------------------------------------------------------------------------
// Errors
//-----------------------------------------------------------------------------
CASE _stStationState.eState
OF
  E_STATION_STATE.STATION_ERROR_LIST_STATION_ID_WRONG:
    IF (_stStationCtrl.eCmd = E_STATION_CTRL.STATION_MOVER_OUT)
    THEN
      _nMoverDetected                 := _stMoverData.nMoverId;

      IF (_nMoverDetected < 1) OR
         (_nMoverDetected > MAX_MOVER)
      THEN
        // this MUST NOT happen
        _stStationState.eState        := E_STATION_STATE.STATION_ERROR_LIST_MOVER_ID_INVALID;
        _stMsg.eType                  := E_MessageType.eMessageError;
        LogState(_stMsg.eType);

      ELSE
        // not for station; send mover out
        _stStationState.eState        := E_STATION_STATE.STATION_MOVER_OUT;

        IF (_eMessageLevel < E_MessageType.eMessageError)
        THEN
          _stMsg.eType                := E_MessageType.eMessageInfo;
          LogState(_stMsg.eType);
        END_IF
      END_IF

    ELSIF (_stStationCtrl.eCmd = E_STATION_CTRL.STATION_MOVER_ENTER)
    THEN
      // override wrong TargetStationId in List; start infeed of mover

      _nMoverDetected                 := _stMoverData.nMoverId;

      IF (_nMoverDetected < 1) OR
         (_nMoverDetected > MAX_MOVER)
      THEN
        // this MUST NOT happen
        _stStationState.eState        := E_STATION_STATE.STATION_ERROR_LIST_MOVER_ID_INVALID;

        _stMsg.eType                  := E_MessageType.eMessageError;
        LogState(_stMsg.eType);

      ELSE
        _eState                       := E_PROGRESS.PROGRESS_INIT;
        _stStationState.nMoverId      := TO_USINT(_nMoverDetected);
        _stStationState.nMask         := _stMoverData.nMask;
        _stStationState.eState        := E_STATION_STATE.STATION_MOVER_ENTER;

        IF (_eMessageLevel < E_MessageType.eMessageError)
        THEN
          _stMsg.eType                := E_MessageType.eMessageInfo;
          LogState(_stMsg.eType);
        END_IF
      END_IF
    END_IF


  E_STATION_STATE.STATION_ERROR_OUTFEED_TARGET_INVALID:
    // wait here until valid target is detected
    IF NOT (_stStationCtrl.nTargetStation < 1) AND  
       NOT (_stStationCtrl.nTargetStation > MAX_STATION)
    THEN
      _stStationState.eState          := E_STATION_STATE.STATION_MOVER_OUT;

      IF (_eMessageLevel < E_MessageType.eMessageError)
      THEN
        _stMsg.eType                  := E_MessageType.eMessageInfo;
        LogState(_stMsg.eType);
      END_IF
    END_IF


  E_STATION_STATE.STATION_ERROR_INFEED_ERROR:   // must be fixed by extern by using cyclic mover control
    IF (_stStationCtrl.eCmd = E_STATION_CTRL.STATION_MOVER_ENTER_RETRY)
    THEN
      _stStationState.eState          := E_STATION_STATE.STATION_DETECT_MOVER;   // return to start and wait

      IF (_eMessageLevel < E_MessageType.eMessageError)
      THEN
        _stMsg.eType                  := E_MessageType.eMessageInfo;
        LogState(_stMsg.eType);
      END_IF
    END_IF


  E_STATION_STATE.STATION_ERROR_OUTFEED_ERROR:  // must be fixed by extern by using cyclic mover control
    IF (_stStationCtrl.eCmd = E_STATION_CTRL.STATION_MOVER_OUT_RETRY)
    THEN
      _stStationState.eState          := E_STATION_STATE.STATION_MOVER_OUT; // return to send out and wait

      IF (_eMessageLevel < E_MessageType.eMessageError)
      THEN
        _stMsg.eType                  := E_MessageType.eMessageInfo;
        LogState(_stMsg.eType);
      END_IF

    ELSIF (_stStationCtrl.eCmd = E_STATION_CTRL.STATION_MOVER_GONE)
    THEN
      MoverOut();

      // add entry in target station list
      _stListTarget                   := _ItfStation[_stMoverDataSend.nTargetStation].AddTailValue(_stMoverDataSend);
      IF (_stListTarget.wState <> 0)
      THEN
        _stStationState.eState        := E_STATION_STATE.STATION_ERROR_LIST_ADD_TAIL_FAULT;
        _stMsg.eType                  := E_MessageType.eMessageError;
        LogState(_stMsg.eType);

      ELSE
        IF (_eMessageLevel < E_MessageType.eMessageError)
        THEN
          _stMsg.eType                := E_MessageType.eMessageInfo;
          _stMsg.eSubdevice           := e_Subdevice.StationAddTail;
          _stMsg.iErrorNumber         := _stStationState.nMoverId;
          _stMsg.sText                := concat('TargetStation: ', TO_STRING(_stListTarget.stData.nTargetStation));
          f_MessageSet(_stMsg);
        END_IF

        _stStationState.eState        := E_STATION_STATE.STATION_MOVER_GONE;

        IF (_eMessageLevel < E_MessageType.eMessageError)
        THEN
          _stMsg.eType                := E_MessageType.eMessageInfo;
          LogState(_stMsg.eType);
        END_IF
      END_IF
    END_IF


  E_STATION_STATE.STATION_ERROR_LIST_GET_HEAD_FAULT,
  E_STATION_STATE.STATION_ERROR_LIST_REMOVE_HEAD_FAULT,
  E_STATION_STATE.STATION_ERROR_LIST_ADD_TAIL_FAULT,
  E_STATION_STATE.STATION_ERROR_LIST_MOVER_ID_INVALID:
    _stMsg.eType                      := E_MessageType.eMessageError;
    LogState(_stMsg.eType);
    // yes, but why?
    // cannot be fixed by ctrl
    _eFatalError                      := _stStationState.eState;
    _stStationState.eState            := E_STATION_STATE.STATION_ERROR_FATAL;

  E_STATION_STATE.STATION_ERROR_FATAL:
    // write to string for debugging
    _sState                           := concat(TO_STRING(_stStationState.eState), ': ');
    _sState                           := concat(_sState, TO_STRING(_eFatalError));
END_CASE

IF (_stStationState.nMoverId <> 0)
THEN
  _stStationState.rMoverModPos        := _Mover[_stStationState.nMoverId].NcToPlc.ModuloActPos;
END_IF

_stStationState.nQueue                := TO_USINT(_ItfStation[_nStationId].Count);
_stState[_nStationId]                 := _stStationState;
END_METHOD

METHOD PUBLIC DelBitWord : WORD
VAR_INPUT
  inVal   : WORD;
  bitNo   : DINT;
END_VAR
VAR
  wConst : WORD := 1;
END_VAR
IF ( inVal AND SHL( wConst,bitNo MOD 16 ) ) > 0 THEN
  DelBitWord := inVal XOR (SHL( wConst,bitNo MOD 16 ));
ELSE
  DelBitWord := inVal;
END_IF
END_METHOD

METHOD PUBLIC GetBitWord : BOOL
VAR_INPUT
  inVal   : WORD;
  bitNo   : DINT;
END_VAR
VAR
  wConst : WORD := 1;
END_VAR
IF ( inVal AND SHL( wConst,DINT_TO_SINT(bitNo) MOD 16 ) ) > 0
THEN
  GetBitWord := TRUE;
ELSE
  GetBitWord := FALSE;
END_IF
END_METHOD

METHOD Init : e_progress
VAR_INPUT
END_VAR
// check pointer and interface
IF NOT Check() THEN Init := e_progress.PROGRESS_ERROR; RETURN; END_IF

_stStationState.nMask             := 0;
_stStationState.nMoverId          := 0;

_eFatalError                      := E_STATION_STATE.STATION_ERROR_NULL;

_stStationState.eState            := E_STATION_STATE.STATION_INIT;
_stState[_nStationId]             := _stStationState;
_sState                           := TO_STRING(_stStationState.eState);

IF _ItfStation[_nStationId].InitList()
THEN
  Init                            := e_progress.PROGRESS_DONE;
ELSE
  Init                            := e_progress.PROGRESS_ERROR;
END_IF
END_METHOD

PROPERTY ItfMover : reference to ARRAY[1..MAX_MOVER] OF I_XtsTransport_Mover
SET
_ItfMover ref= ItfMover;
END_SET
END_PROPERTY

PROPERTY ItfStations : reference to ARRAY[1..MAX_STATION] OF I_Station_LinkedList
SET
_ItfStation ref= ItfStations;
END_SET
END_PROPERTY

METHOD LogState
VAR_INPUT
  eType       : E_MessageType;
END_VAR
_stMsg.eType                := eType;
_stMsg.eSubdevice           := Stationstate;
_stMsg.iErrorNumber         := _stStationState.nMoverId;
_stMsg.sText                := TO_STRING(_stStationState.eState);
f_MessageSet(_stMsg);
END_METHOD

PROPERTY MessageLevel : e_messagetype
SET
_eMessageLevel := MessageLevel;
END_SET
END_PROPERTY

METHOD PRIVATE MoveData
// build WorkPos from parameter, static station data and information on mover
_stInfeed.rPos            := TO_REAL(_stParameter[_nStationId].rPosWait
                             + _stParameter[_nStationId].rPosStop[_nNest]
                             + _stMoverData.rOffset
                             + _rMoverOffset[_nStationId][_stMoverData.nMoverId][_nNest]);

_stInfeed.rVelo           := _stParameter[_nStationId].rVelo;
_stInfeed.rAcc            := _stParameter[_nStationId].rAccDec;
_stInfeed.rJerk           := _stParameter[_nStationId].rJerk;
_stInfeed.rGap            := _stParameter[_nStationId].rGap;
_stInfeed.rDistance       := _stParameter[_nStationId].rReleaseDistance;

// init method and state
_ItfMover[_stMoverData.nMoverId].MoveToPosCa(FALSE, _stInfeed);
_eState                     := E_PROGRESS.PROGRESS_INIT;
END_METHOD

PROPERTY Mover : reference TO ARRAY[1..MAX_MOVER] OF AXIS_REF;
SET
_Mover ref= Mover;
END_SET
END_PROPERTY

PROPERTY MoverOffset : reference TO ARRAY[1..MAX_STATION]  OF T_NEST_OFFSET
SET
_rMoverOffset ref= MoverOffset;
END_SET
END_PROPERTY

METHOD PRIVATE MoverOut
VAR_INPUT
END_VAR
// build data for sending mover to target station

// who am I sending?
_stMoverDataSend.nMoverId         := _stStationState.nMoverId;

// get optional information about nests to work
_stMoverDataSend.nMask            := _stStationCtrl.nMask;

// get optional offset
_stMoverDataSend.rOffset          := _stStationCtrl.rOffset;

// get target station
_stMoverDataSend.nTargetStation   := _stStationCtrl.nTargetStation;

// get position of target
_stOutfeed.rPos               := TO_REAL(_stParameter[_stMoverDataSend.nTargetStation].rPosWait);

IF (_stOutfeed.rPos - TO_REAL(_Mover[_stMoverDataSend.nMoverId].NcToPlc.ModuloActPos) < 0)
THEN
  // only forward, never back
  _stOutfeed.rPos             := TO_REAL(_stOutfeed.rPos 
                                 + _ItfMover[_stMoverDataSend.nMoverId].RailLength);
END_IF

_stOutfeed.rVelo              := _stParameter[_nStationId].rVelo;
_stOutfeed.rAcc               := _stParameter[_nStationId].rAccDec;
_stOutfeed.rJerk              := _stParameter[_nStationId].rJerk;
_stOutfeed.rGap               := _stParameter[_nStationId].rGap;
_stOutfeed.rDistance          := _stParameter[_nStationId].rReleaseDistance;

// init method for sending
_ItfMover[_stMoverDataSend.nMoverId].SendToModuloPosCa(FALSE, 
                                                  _stOutfeed);
END_METHOD

METHOD PUBLIC SetBitWord : WORD
VAR_INPUT
  inVal   : WORD;
  bitNo   : DINT;
END_VAR
VAR
  wConst  : WORD := 1;
END_VAR
SetBitWord := inVal OR SHL( wConst,bitNo MOD 16 );
END_METHOD

PROPERTY State : reference to ARRAY[1..MAX_STATION] OF ST_STATION_STATE
SET
_stState ref= State;
END_SET
END_PROPERTY

PROPERTY StationId : uint
GET
StationId := _nStationId;
END_GET
SET
_nStationId := StationId;
END_SET
END_PROPERTY

PROPERTY StationParameter : reference TO ARRAY[1..MAX_STATION]  OF ST_STATION_PARAMETER
SET
_stParameter ref= StationParameter;
END_SET
END_PROPERTY

END_FUNCTION_BLOCK

// ---- XTS/XtsTransportUnit/fb_TransportUnit.TcPOU
//---------------------------------------------------------------------------------------------------------------
//
//  HAUD 2024.03.18
//
//  - XTS_TRANSPORT_LAYER
//
//  fb_TransportUnit
//  - Ctrl/STate interface, reacts to change of command
//    - Cmd(E_TRANSPORT_CTRL)
//
//  - controls members via structures and interfaces for getting XTS in defined state
//    - CMD_INIT:
//        - XPU is initialized:         XTS_CMD_INIT + PROGRESS_DONE
//        - XPU cyclic checks enabled:  XTS_IDLE     + PROGRESS_WORKING
//        - XPU detects mover:          _XpuState.Check == MOVER_ID_DETECTION_VALID
//
//    - CMD_IDLE
//      - Cyclic Checks of XPU and CaGroup
//        - XPU cyclic checks enabled:  XTS_IDLE     + PROGRESS_WORKING
//
//
//  CTRL / STATE --> see proprerties
//  structs for use of function block via mapping
//  cyclic check for new command
//
//  VAR INPUT / OUTPUT --> see properties
//
//---------------------------------------------------------------------------------------------------------------
// This SOFTWARE is provided as an Exemple by THE PROVIDER "as is" and "with all faults." THE PROVIDER makes no 
// representations or warranties of any kind concerning the safety, suitability, lack of viruses, inaccuracies, 
// typographical errors, or other harmful components of this SOFTWARE. There are inherent dangers in the use of 
// any software, and you are solely responsible for determining whether this SOFTWARE is compatible with your 
// equipment and other software installed on your equipment. You are also solely responsible for the protection 
// of your equipment and backup of your data, and THE PROVIDER will not be liable for any damages you may suffer 
// in connection with using, modifying, or distributing this SOFTWARE.
//---------------------------------------------------------------------------------------------------------------
FUNCTION_BLOCK fb_TransportUnit
VAR
  _eCheck                       : E_XTS_TRANSPORT_CHECK;

  // Transport Ctrl/State
  _Ctrl                         : REFERENCE TO ST_XTS_TRANSPORT_CTRL;
  _State                        : REFERENCE TO ST_XTS_TRANSPORT_STATE;


  // execute transport commands
  _eCmd,
  _eCmdOld                      : E_XTS_TRANSPORT_CTRL;

  // execution state
  _eState                       : E_XTS_TRANSPORT_STATE;

  // execution result
  _eJobResult,
  _eResult                      : E_PROGRESS;


  // members of transport
  _XpuCtrl                      : REFERENCE TO ST_XPU_CTRL;                     // processing unit ctrl
  _XpuState                     : REFERENCE TO ST_XPU_STATE;                    // processing unit state
  _XpuInfo                      : REFERENCE TO ST_XPU_INFO;                     // processing unit information

  _GroupItf                     : I_XtsTransport_CaGroup;                       // group methods
  _GroupInfo                    : REFERENCE TO ST_GROUP_INFO;                   // info from group

  _MoverItf                     : REFERENCE TO ARRAY[1..MAX_MOVER] OF I_XtsTransport_Mover;  // mover methods
  _MoverInfo                    : REFERENCE TO ARRAY[1..MAX_MOVER] OF ST_MOVER_INFO;         // info from mover

  _StationStart                 : REFERENCE TO ST_STATION_PARAMETER;            // position, gap, dynamic constraints for sending all mover to start position

  // stations lists
  _ItfStationList               : REFERENCE TO ARRAY[1..MAX_STATION]  OF I_Station_LinkedList;  // access to all stations lists

  // access to stations methods by interface
  _ItfStationCtrl               : REFERENCE TO ARRAY[1..MAX_STATION]  OF I_XtsTransport_Station;

  _nStartStation                : UINT;

  _stMoverDataSend              : ST_STATION_MOVER_DATA;    // mover ticket data

  _stListResult                 : ST_STATION_LIST_RESULT;
END_VAR

IF NOT Check() THEN RETURN; END_IF

_eCmd                         := _Ctrl.Cmd;

// check for command change
// get state for cmd
IF (_eCmd <> _eCmdOld)
THEN
  _eState                     := Cmd(_eCmd);
  _eCmdOld                    := _eCmd;
END_IF


CASE _eState
OF
  E_XTS_TRANSPORT_STATE.TRANSPORT_INIT:
    _eResult                  := XpuInit(TRUE);

  E_XTS_TRANSPORT_STATE.TRANSPORT_IDLE:
    _eResult                  := f_GetProgress(_XpuState.State);

    IF (_GroupInfo.GroupErrorStop) OR
       (_GroupInfo.GroupError)
    THEN
      _eResult                := E_PROGRESS.PROGRESS_ERROR;
    END_IF

  E_XTS_TRANSPORT_STATE.TRANSPORT_MOVER_ENABLE:
    _eResult                  := MoverEnableAll(TRUE);

  E_XTS_TRANSPORT_STATE.TRANSPORT_MOVER_DISABLE:
    _eResult                  := MoverDisableAll(TRUE);

  E_XTS_TRANSPORT_STATE.TRANSPORT_GROUP_CLEAR:
    _eResult                  := GroupClear(TRUE);

  E_XTS_TRANSPORT_STATE.TRANSPORT_GROUP_BUILD:
    _eResult                  := GroupBuild(TRUE);

  E_XTS_TRANSPORT_STATE.TRANSPORT_GROUP_ENABLE:
    _eResult                  := GroupEnable(TRUE);

  E_XTS_TRANSPORT_STATE.TRANSPORT_START:
    _eResult                  := TransportStart(TRUE);

  E_XTS_TRANSPORT_STATE.TRANSPORT_RESTART:
    _eResult                  := TransportRestart(TRUE);

ELSE
  _eResult                    := E_PROGRESS.PROGRESS_INVALID;
END_CASE


CASE _eResult
OF
  E_PROGRESS.PROGRESS_INVALID:
    _State.State              := TO_UINT(_eResult);

  E_PROGRESS.PROGRESS_ERROR:
    _State.State              := _eState + E_PROGRESS.PROGRESS_ERROR;

  E_PROGRESS.PROGRESS_DONE:
    _State.State              := _eState + E_PROGRESS.PROGRESS_DONE;

ELSE
  _State.State                := _eState + _eResult;
END_CASE

_State.XpuState               := _XpuState;
_State.XpuInfo                := _XpuInfo;
_State.GroupInfo              := _GroupInfo;

METHOD PRIVATE Check  : BOOL
VAR_INST
  _idx        : UINT;
END_VAR

IF NOT __ISVALIDREF(_Ctrl)
THEN
  _eCheck                     := E_XTS_TRANSPORT_CHECK.POINTER_NULL_CTRL;
  RETURN;
END_IF

IF NOT __ISVALIDREF(_State)
THEN
  _eCheck                     := E_XTS_TRANSPORT_CHECK.POINTER_NULL_STATE;
  RETURN;
END_IF

_State.Check                  := _eCheck;

IF NOT __ISVALIDREF(_XpuCtrl)
THEN
  _eCheck                     := E_XTS_TRANSPORT_CHECK.POINTER_NULL_XPU_CTRL;
  RETURN;
END_IF

IF NOT __ISVALIDREF(_XpuState)
THEN
  _eCheck                     := E_XTS_TRANSPORT_CHECK.POINTER_NULL_XPU_STATE;
  RETURN;
END_IF

IF NOT __ISVALIDREF(_XpuInfo)
THEN
  _eCheck                     := E_XTS_TRANSPORT_CHECK.POINTER_NULL_XPU_INFO;
  RETURN;
END_IF

IF NOT (_GroupItf <> 0)
THEN
  _eCheck                     := E_XTS_TRANSPORT_CHECK.POINTER_NULL_GROUP_ITF;
  RETURN;
END_IF

IF NOT __ISVALIDREF(_GroupInfo)
THEN
  _eCheck                     := E_XTS_TRANSPORT_CHECK.POINTER_NULL_GROUP_INFO;
  RETURN;
END_IF

IF NOT __ISVALIDREF(_MoverItf)
THEN
  _eCheck                     := E_XTS_TRANSPORT_CHECK.POINTER_NULL_MOVER;
  RETURN;
END_IF

FOR _idx := 1 TO MAX_MOVER
DO
  IF NOT (_MoverItf[_idx] <> 0)
  THEN
    _eCheck                   := E_XTS_TRANSPORT_CHECK.POINTER_NULL_MOVER_ITF;
    RETURN;
  END_IF
END_FOR

IF NOT __ISVALIDREF(_MoverInfo)
THEN
  _eCheck                     := E_XTS_TRANSPORT_CHECK.POINTER_NULL_MOVER_INFO;
  RETURN;
END_IF

IF NOT __ISVALIDREF(_StationStart)
THEN
  _eCheck                     := E_XTS_TRANSPORT_CHECK.POINTER_NULL_STATION_START;
  RETURN;
END_IF

IF NOT __ISVALIDREF(_ItfStationList)
THEN
  _eCheck                     := E_XTS_TRANSPORT_CHECK.POINTER_NULL_STATION_ITF;
  RETURN;
END_IF

IF NOT __ISVALIDREF(_ItfStationCtrl)
THEN
  _eCheck                     := E_XTS_TRANSPORT_CHECK.POINTER_NULL_STATION_CTRL;
  RETURN;
END_IF


_eCheck                       := E_XTS_TRANSPORT_CHECK.DONE_CHECK;
Check                         := TRUE;
END_METHOD

METHOD PRIVATE Cmd : E_XTS_TRANSPORT_STATE
VAR_INPUT
  Ctrl      : E_XTS_TRANSPORT_CTRL;
END_VAR
VAR_INST
  _eRslt    : E_PROGRESS;
  _eState   : E_XTS_TRANSPORT_STATE;
  _eCk      : E_XTS_TRANSPORT_CHECK;
END_VAR
IF NOT Check() THEN RETURN; END_IF


CASE Ctrl
OF
  E_XTS_TRANSPORT_CTRL.CMD_NULL:  // clear all method calls
    _eState               := E_XTS_TRANSPORT_STATE.TRANSPORT_NULL;
    _eRslt                := XpuInit         (FALSE);
    _eRslt                := GroupClear      (FALSE);
    _eRslt                := GroupBuild      (FALSE);
    _eRslt                := GroupEnable     (FALSE);
    _eRslt                := MoverEnableAll  (FALSE);
    _eRslt                := MoverDisableAll (FALSE);
    _eRslt                := TransportRestart(FALSE);
    _eRslt                := TransportRestart(FALSE);

  E_XTS_TRANSPORT_CTRL.CMD_INIT:  // clear methods for initialization
    _eState               := E_XTS_TRANSPORT_STATE.TRANSPORT_INIT;
    _eResult              := XpuInit(FALSE);


ELSE
  IF NOT (_XpuState.Init = E_XPU_INIT.INIT_DONE)
  THEN
    // no init, no further commands possible
    _eState               := E_XTS_TRANSPORT_STATE.TRANSPORT_INVALID;
  ELSE
    CASE Ctrl
    OF
      E_XTS_TRANSPORT_CTRL.CMD_IDLE:
        _eState           := E_XTS_TRANSPORT_STATE.TRANSPORT_IDLE;

      E_XTS_TRANSPORT_CTRL.CMD_MOVER_ENABLE:
        _eState           := E_XTS_TRANSPORT_STATE.TRANSPORT_MOVER_ENABLE;
        _eResult          := MoverEnableAll(FALSE);

      E_XTS_TRANSPORT_CTRL.CMD_MOVER_DISABLE:
        _eState           := E_XTS_TRANSPORT_STATE.TRANSPORT_MOVER_DISABLE;
        _eResult          := MoverDisableAll(FALSE);

      E_XTS_TRANSPORT_CTRL.CMD_GROUP_CLEAR:
        _eState           := E_XTS_TRANSPORT_STATE.TRANSPORT_GROUP_CLEAR;
        _eResult          := GroupClear (FALSE);

      E_XTS_TRANSPORT_CTRL.CMD_GROUP_BUILD:
        _eState           := E_XTS_TRANSPORT_STATE.TRANSPORT_GROUP_BUILD;
        _eResult          := GroupBuild (FALSE);

      E_XTS_TRANSPORT_CTRL.CMD_GROUP_ENABLE:
        _eState           := E_XTS_TRANSPORT_STATE.TRANSPORT_GROUP_ENABLE;
        _eResult          := GroupEnable(FALSE);

      E_XTS_TRANSPORT_CTRL.CMD_TRANSPORT_START:
        _eState           := E_XTS_TRANSPORT_STATE.TRANSPORT_START;
        _eResult          := TransportStart(FALSE);

      E_XTS_TRANSPORT_CTRL.CMD_TRANSPORT_RESTART:
        _eState           := E_XTS_TRANSPORT_STATE.TRANSPORT_RESTART;
        _eResult          := TransportRestart(FALSE);

    ELSE
        _eState           := E_XTS_TRANSPORT_STATE.TRANSPORT_INVALID;
    END_CASE
  END_IF
END_CASE

Cmd                       := _eState;
END_METHOD

PROPERTY Ctrl : REFERENCE TO ST_XTS_TRANSPORT_CTRL
SET
_Ctrl REF= Ctrl;
END_SET
END_PROPERTY

METHOD GroupBuild : E_PROGRESS
VAR_INPUT
  Execute     : BOOL;
END_VAR
VAR_INST
  _nErrorId   : UDINT;
  _eJobReslt,
  _eState     : E_PROGRESS;
END_VAR
//-----------------------------------------------------------------------------
IF NOT Execute 
THEN 
	_eState                       := E_PROGRESS.PROGRESS_INIT; 
END_IF 
//-----------------------------------------------------------------------------
IF NOT Check() 
THEN 
	GroupBuild                    := E_PROGRESS.PROGRESS_ERROR; 
	RETURN; 
END_IF
//-----------------------------------------------------------------------------
//-----------------------------------------------------------------------------
CASE _eState
OF
  E_PROGRESS.PROGRESS_INIT:
    IF Execute
    THEN
      _nErrorId                 := 0;

      IF (_GroupInfo.AxisCount <> 0)
      THEN
        _nErrorId               := 9999;
        _eState                 := E_PROGRESS.PROGRESS_ERROR;
      ELSE
        _eState                 := E_PROGRESS.PROGRESS_BUSY;
        _eJobReslt              := _GroupItf.AddAll(FALSE);
      END_IF
    END_IF
END_CASE
//---------------------------------------------------------------------------
//---------------------------------------------------------------------------
CASE _eState
OF
  E_PROGRESS.PROGRESS_BUSY:
    _eJobReslt                  := _GroupItf.AddAll(TRUE);

    IF (_eJobReslt = E_PROGRESS.PROGRESS_ERROR)
    THEN
      _eState                   := E_PROGRESS.PROGRESS_ERROR;

      _nErrorId                 := _GroupInfo.GroupErrorId;
      _eJobReslt                := _GroupItf.AddAll(FALSE);

    ELSIF (_eJobReslt = E_PROGRESS.PROGRESS_DONE)
    THEN
      _eState                   := E_PROGRESS.PROGRESS_DONE;
      _eJobReslt                := _GroupItf.AddAll(FALSE);
    END_IF
END_CASE
//-----------------------------------------------------------------------------
//-----------------------------------------------------------------------------

GroupBuild                      := _eState;
END_METHOD

METHOD GroupClear : E_PROGRESS
VAR_INPUT
  Execute     : BOOL;
END_VAR
VAR_INST
  _nErrorId   : UDINT;
  _eJobReslt,
  _eState     : E_PROGRESS;
END_VAR
//-----------------------------------------------------------------------------
IF NOT Execute 
THEN 
	_eState                       := E_PROGRESS.PROGRESS_INIT; 
END_IF 
//-----------------------------------------------------------------------------
IF NOT Check() 
THEN 
	GroupClear                    := E_PROGRESS.PROGRESS_ERROR; 
	RETURN; 
END_IF
//-----------------------------------------------------------------------------
//-----------------------------------------------------------------------------
CASE _eState
OF
  E_PROGRESS.PROGRESS_INIT:
    IF Execute
    THEN
      _nErrorId                 := 0;
      _eJobReslt                := _GroupItf.McHaltAll(FALSE);
      _eState                   := E_PROGRESS.PROGRESS_BUSY;
    END_IF
  //---------------------------------------------------------------------------
  //---------------------------------------------------------------------------
  E_PROGRESS.PROGRESS_BUSY:
    _eJobReslt                  := _GroupItf.McHaltAll(TRUE);

    IF (_eJobReslt = E_PROGRESS.PROGRESS_ERROR)
    THEN
      _eState                   := E_PROGRESS.PROGRESS_ERROR;
      _nErrorId                 := _GroupInfo.GroupErrorId;
      _eJobReslt                := _GroupItf.McHaltAll(FALSE);

    ELSIF (_eJobReslt = E_PROGRESS.PROGRESS_DONE)
    THEN
      _eState                   := E_PROGRESS.PROGRESS_PREPARE;
      _eJobReslt                := _GroupItf.McResetAll(FALSE);
      _eJobReslt                := _GroupItf.McHaltAll(FALSE);
    END_IF
  //---------------------------------------------------------------------------
  //---------------------------------------------------------------------------
  E_PROGRESS.PROGRESS_PREPARE:
    _eJobReslt                  := _GroupItf.McResetAll(TRUE);

    IF (_eJobReslt = E_PROGRESS.PROGRESS_ERROR)
    THEN
      _eState                   := E_PROGRESS.PROGRESS_ERROR;
      _nErrorId                 := _GroupInfo.GroupErrorId;
      _eJobReslt                := _GroupItf.McResetAll(FALSE);

    ELSIF (_eJobReslt = E_PROGRESS.PROGRESS_DONE)
    THEN
      _eState                   := E_PROGRESS.PROGRESS_STARTUP;
      _eJobReslt                := _GroupItf.McResetAll(FALSE);
      _eJobReslt                := _GroupItf.RemoveAll(FALSE);
    END_IF
  //---------------------------------------------------------------------------
  //---------------------------------------------------------------------------
  E_PROGRESS.PROGRESS_STARTUP:
    _eJobReslt                  := _GroupItf.RemoveAll(TRUE);

    IF (_eJobReslt = E_PROGRESS.PROGRESS_ERROR)
    THEN
      _eState                   := E_PROGRESS.PROGRESS_ERROR;
      _nErrorId                 := _GroupInfo.GroupErrorId;
      _eJobReslt                := _GroupItf.RemoveAll(FALSE);

    ELSIF (_eJobReslt = E_PROGRESS.PROGRESS_DONE)
    THEN
      _eState                   := E_PROGRESS.PROGRESS_CHECK;
      _eJobReslt                := _GroupItf.RemoveAll(FALSE);
      _eJobReslt                := _GroupItf.Disable(FALSE);
    END_IF
  //---------------------------------------------------------------------------
  //---------------------------------------------------------------------------
  E_PROGRESS.PROGRESS_CHECK:
    _eJobReslt                  := _GroupItf.Disable(TRUE);

    IF (_eJobReslt = E_PROGRESS.PROGRESS_ERROR)
    THEN
      _eState                   := E_PROGRESS.PROGRESS_ERROR;
      _nErrorId                 := _GroupInfo.GroupErrorId;
      _eJobReslt                := _GroupItf.Disable(FALSE);

    ELSIF (_eJobReslt = E_PROGRESS.PROGRESS_DONE)
    THEN
      _eState                   := E_PROGRESS.PROGRESS_OCCUPIED;
      _eJobReslt                := _GroupItf.Disable(FALSE);
      _eJobReslt                := _GroupItf.Reset(FALSE);
    END_IF
  //---------------------------------------------------------------------------
  //---------------------------------------------------------------------------
  E_PROGRESS.PROGRESS_OCCUPIED:
    _eJobReslt                 := _GroupItf.Reset(TRUE);

    IF (_eJobReslt = E_PROGRESS.PROGRESS_ERROR)
    THEN
      _eState                   := E_PROGRESS.PROGRESS_ERROR;
      _nErrorId                 := _GroupInfo.GroupErrorId;
      _eJobReslt                := _GroupItf.Reset(FALSE);

    ELSIF (_eJobReslt = E_PROGRESS.PROGRESS_DONE)
    THEN
      _eState                   := E_PROGRESS.PROGRESS_WORKING;
      _eJobReslt                := _GroupItf.Reset(FALSE);
    END_IF
END_CASE
//-----------------------------------------------------------------------------
//-----------------------------------------------------------------------------
CASE _eState
OF
  E_PROGRESS.PROGRESS_WORKING:
    IF (_GroupInfo.GroupDisabled) AND NOT
       (_GroupInfo.GroupError)
    THEN
      _eState                   := E_PROGRESS.PROGRESS_DONE;
    ELSE
      IF (_GroupInfo.GroupErrorStop) OR
         (_GroupInfo.GroupError)
      THEN
        _eState                 := E_PROGRESS.PROGRESS_ERROR;
      END_IF
    END_IF
END_CASE
//-----------------------------------------------------------------------------
//-----------------------------------------------------------------------------

GroupClear                      := _eState;
END_METHOD

METHOD GroupEnable : E_PROGRESS
VAR_INPUT
  Execute     : BOOL;
END_VAR
VAR_INST
  _nErrorId   : UDINT;
  _eJobReslt,
  _eState     : E_PROGRESS;
END_VAR
//-----------------------------------------------------------------------------
IF NOT Execute 
THEN 
	_eState                       := E_PROGRESS.PROGRESS_INIT; 
END_IF 
//-----------------------------------------------------------------------------
IF NOT Check() 
THEN 
	GroupEnable                   := E_PROGRESS.PROGRESS_ERROR; 
	RETURN; 
END_IF
//-----------------------------------------------------------------------------
//-----------------------------------------------------------------------------
CASE _eState
OF
  E_PROGRESS.PROGRESS_INIT:
    IF Execute
    THEN
      _nErrorId                 := 0;

      IF NOT (_GroupInfo.AxisCount <> 0)
      THEN
        _nErrorId               := 9999;
        _eState                 := E_PROGRESS.PROGRESS_ERROR;
      ELSE
        _eState                 := E_PROGRESS.PROGRESS_BUSY;
        _eJobReslt              := _GroupItf.Enable(FALSE);
      END_IF
    END_IF
END_CASE
//---------------------------------------------------------------------------
//---------------------------------------------------------------------------
CASE _eState
OF
  E_PROGRESS.PROGRESS_BUSY:
    _eJobReslt                  := _GroupItf.Enable(TRUE);

    IF (_eJobReslt = E_PROGRESS.PROGRESS_ERROR)
    THEN
      _eState                   := E_PROGRESS.PROGRESS_ERROR;

      _nErrorId                 := _GroupInfo.GroupErrorId;
      _eJobReslt                := _GroupItf.Enable(FALSE);

    ELSIF (_eJobReslt = E_PROGRESS.PROGRESS_DONE)
    THEN
      _eState                   := E_PROGRESS.PROGRESS_CHECK;
      _eJobReslt                := _GroupItf.Enable(FALSE);
    END_IF
END_CASE
//-----------------------------------------------------------------------------
//-----------------------------------------------------------------------------
CASE _eState
OF
  E_PROGRESS.PROGRESS_CHECK:
    IF (_GroupInfo.GroupStandby) OR
       (_GroupInfo.GroupMoving)  OR
       (_GroupInfo.GroupNotReady)
    THEN
      _eState                   := E_PROGRESS.PROGRESS_DONE;
    ELSE
      IF (_GroupInfo.GroupErrorStop) OR
         (_GroupInfo.GroupError)
      THEN
        _eState                 := E_PROGRESS.PROGRESS_ERROR;
      END_IF
    END_IF
END_CASE
//-----------------------------------------------------------------------------
//-----------------------------------------------------------------------------
GroupEnable                     := _eState;
END_METHOD

PROPERTY GroupInfo : REFERENCE TO ST_GROUP_INFO
SET
_GroupInfo REF= GroupInfo;
END_SET
END_PROPERTY

PROPERTY GroupItf : I_XtsTransport_CaGroup
SET
_GroupItf := GroupItf;
END_SET
END_PROPERTY

METHOD MoverDisableAll : e_progress
VAR_INPUT
  Execute     : BOOL;
END_VAR
VAR_INST
  _nMover     : UINT;
  _nErrorId   : UDINT;
  _eRslt,
  _eState     : E_PROGRESS;
END_VAR
//-----------------------------------------------------------------------------
IF NOT Execute 
THEN 
	_eState                       := E_PROGRESS.PROGRESS_INIT; 
END_IF 
//-----------------------------------------------------------------------------
IF NOT Check() 
THEN 
	MoverDisableAll               := E_PROGRESS.PROGRESS_ERROR; 
	RETURN; 
END_IF
//-----------------------------------------------------------------------------
//-----------------------------------------------------------------------------
CASE _eState
OF
  E_PROGRESS.PROGRESS_INIT:
    IF Execute
    THEN
      _nErrorId                 := 0;
      _nMover                   := 1;

      _eState                   := E_PROGRESS.PROGRESS_BUSY;
    END_IF
END_CASE
//-----------------------------------------------------------------------------
//-----------------------------------------------------------------------------
CASE _eState
OF
  E_PROGRESS.PROGRESS_BUSY:
    _eState                     := E_PROGRESS.PROGRESS_PREPARE;
    _eRslt                      := _MoverItf[_nMover].Disable(FALSE);
END_CASE
//-----------------------------------------------------------------------------
//-----------------------------------------------------------------------------
CASE _eState
OF
  E_PROGRESS.PROGRESS_PREPARE:
    _eRslt                      := _MoverItf[_nMover].Disable(TRUE);

    IF (_eRslt = E_PROGRESS.PROGRESS_ERROR)
    THEN
      _eState                   := E_PROGRESS.PROGRESS_ERROR;
      _nErrorId                 := _MoverInfo[_nMover].nErrorId; 

    ELSIF (_eRslt = E_PROGRESS.PROGRESS_DONE)
    THEN
      _eState                   := E_PROGRESS.PROGRESS_STARTUP;
    END_IF
END_CASE
//-----------------------------------------------------------------------------
//-----------------------------------------------------------------------------
CASE _eState
OF
  E_PROGRESS.PROGRESS_STARTUP:
    _eState                     := E_PROGRESS.PROGRESS_CHECK;
    _eRslt                      := _MoverItf[_nMover].Disable(FALSE);
END_CASE
//-----------------------------------------------------------------------------
//-----------------------------------------------------------------------------
CASE _eState
OF
  E_PROGRESS.PROGRESS_CHECK:
    IF (_nMover > MAX_MOVER-1)
    THEN
      _eState                   := E_PROGRESS.PROGRESS_DONE;
    ELSE
      _nMover                   := _nMover + 1;
      _eState                   := E_PROGRESS.PROGRESS_BUSY;
    END_IF
END_CASE
//-----------------------------------------------------------------------------
//-----------------------------------------------------------------------------

MoverDisableAll                 := _eState;
END_METHOD

METHOD MoverEnableAll : e_progress
VAR_INPUT
  Execute     : BOOL;
END_VAR
VAR_INST
  _nMover     : UINT;
  _nErrorId   : UDINT;
  _eRslt,
  _eState     : E_PROGRESS;
END_VAR
//-----------------------------------------------------------------------------
IF NOT Execute 
THEN 
	_eState                       := E_PROGRESS.PROGRESS_INIT; 
END_IF 
//-----------------------------------------------------------------------------
IF NOT Check() 
THEN 
	MoverEnableAll                := E_PROGRESS.PROGRESS_ERROR; 
	RETURN; 
END_IF
//-----------------------------------------------------------------------------
//-----------------------------------------------------------------------------
CASE _eState
OF
  E_PROGRESS.PROGRESS_INIT:
    IF Execute
    THEN
      _nErrorId                 := 0;
      _nMover                   := 1;

      _eState                   := E_PROGRESS.PROGRESS_BUSY;
    END_IF
END_CASE
//-----------------------------------------------------------------------------
//-----------------------------------------------------------------------------
CASE _eState
OF
  E_PROGRESS.PROGRESS_BUSY:
    _eState                     := E_PROGRESS.PROGRESS_PREPARE;
    _eRslt                      := _MoverItf[_nMover].Enable(FALSE);
END_CASE
//-----------------------------------------------------------------------------
//-----------------------------------------------------------------------------
CASE _eState
OF
  E_PROGRESS.PROGRESS_PREPARE:
    _eRslt                      := _MoverItf[_nMover].Enable(TRUE);

    IF (_eRslt = E_PROGRESS.PROGRESS_ERROR)
    THEN
      _eState                   := E_PROGRESS.PROGRESS_ERROR;
      _nErrorId                 := _MoverInfo[_nMover].nErrorId; 

    ELSIF (_eRslt = E_PROGRESS.PROGRESS_DONE)
    THEN
      _eState                   := E_PROGRESS.PROGRESS_STARTUP;
    END_IF
END_CASE
//-----------------------------------------------------------------------------
//-----------------------------------------------------------------------------
CASE _eState
OF
  E_PROGRESS.PROGRESS_STARTUP:
    _eState                     := E_PROGRESS.PROGRESS_CHECK;
    _eRslt                      := _MoverItf[_nMover].Enable(FALSE);
END_CASE
//-----------------------------------------------------------------------------
//-----------------------------------------------------------------------------
CASE _eState
OF
  E_PROGRESS.PROGRESS_CHECK:
    IF (_nMover > MAX_MOVER-1)
    THEN
      _eState                   := E_PROGRESS.PROGRESS_DONE;
    ELSE
      _nMover                   := _nMover + 1;
      _eState                   := E_PROGRESS.PROGRESS_BUSY;
    END_IF
END_CASE
//-----------------------------------------------------------------------------
//-----------------------------------------------------------------------------

MoverEnableAll                  := _eState;
END_METHOD

PROPERTY MoverInfo : REFERENCE TO ARRAY[1..MAX_MOVER] OF ST_MOVER_INFO
SET
_MoverInfo REF= MoverInfo;
END_SET
END_PROPERTY

PROPERTY MoverItf : reference TO ARRAY[1..MAX_MOVER] OF I_XtsTransport_Mover
SET
_MoverItf REF= MoverItf;
END_SET
END_PROPERTY

PROPERTY StartStationIndex : uint
GET
StartStationIndex := _nStartStation;
END_GET
SET
_nStartStation := StartStationIndex;
END_SET
END_PROPERTY

PROPERTY State : REFERENCE TO ST_XTS_TRANSPORT_STATE
SET
_State ref= State;
END_SET
END_PROPERTY

PROPERTY StationCtrlItf : REFERENCE TO ARRAY[1..MAX_STATION]  OF I_XtsTransport_Station;
SET
_ItfStationCtrl REF= StationCtrlItf;
END_SET
END_PROPERTY

PROPERTY StationListsItf : reference to ARRAY[1..MAX_STATION] OF I_Station_LinkedList
SET
_ItfStationList ref= StationListsItf;
END_SET
END_PROPERTY

PROPERTY StationStart : reference to ST_STATION_PARAMETER
SET
_StationStart REF= StationStart;
END_SET
END_PROPERTY

METHOD Template : E_PROGRESS
VAR_INPUT
  Execute     : BOOL;
END_VAR
VAR_INST
  _nErrorId   : UDINT;
  _eState     : E_PROGRESS;
END_VAR
//-----------------------------------------------------------------------------
IF NOT Execute 
THEN 
	_eState                       := E_PROGRESS.PROGRESS_INIT; 
END_IF 
//-----------------------------------------------------------------------------
IF NOT Check() 
THEN 
	Template_1                    := E_PROGRESS.PROGRESS_ERROR; 
	RETURN; 
END_IF
//-----------------------------------------------------------------------------
//-----------------------------------------------------------------------------
CASE _eState
OF
  E_PROGRESS.PROGRESS_INIT:
    IF Execute
    THEN
      _nErrorId                 := 0;

      _eState                   := E_PROGRESS.PROGRESS_BUSY;
    END_IF
END_CASE
//-----------------------------------------------------------------------------
//-----------------------------------------------------------------------------
CASE _eState
OF
  E_PROGRESS.PROGRESS_BUSY:
    _eState                     := E_PROGRESS.PROGRESS_PREPARE;
END_CASE
//-----------------------------------------------------------------------------
//-----------------------------------------------------------------------------
CASE _eState
OF
  E_PROGRESS.PROGRESS_PREPARE:

    IF (.Error)
    THEN
      _eState                   := E_PROGRESS.PROGRESS_ERROR;
      _nErrorId                 := 


    ELSIF (.Done)
    THEN
      _eState                   := E_PROGRESS.;

    END_IF
END_CASE
//-----------------------------------------------------------------------------
//-----------------------------------------------------------------------------

Template_1                      := _eState;
END_METHOD

METHOD TransportRestart : e_progress
VAR_INPUT
  Execute     : BOOL;
END_VAR
VAR_INST
  _nMover     : UINT;
  _nErrorId   : UDINT;
  _eRslt,
  _eState     : E_PROGRESS;
END_VAR
//-----------------------------------------------------------------------------
IF NOT Execute 
THEN 
	_eState                       := E_PROGRESS.PROGRESS_INIT; 
END_IF 
//-----------------------------------------------------------------------------
IF NOT Check() 
THEN 
	TransportRestart              := E_PROGRESS.PROGRESS_ERROR; 
	RETURN; 
END_IF
//-----------------------------------------------------------------------------
//-----------------------------------------------------------------------------
CASE _eState
OF
  E_PROGRESS.PROGRESS_INIT:
    IF Execute
    THEN
      _nErrorId                 := 0;
      _nMover                   := 1;

      _eState                   := E_PROGRESS.PROGRESS_BUSY;
    END_IF
END_CASE
//-----------------------------------------------------------------------------
//-----------------------------------------------------------------------------
CASE _eState
OF
  E_PROGRESS.PROGRESS_BUSY:
    _eState                     := E_PROGRESS.PROGRESS_PREPARE;

END_CASE
//-----------------------------------------------------------------------------
//-----------------------------------------------------------------------------
CASE _eState
OF
  E_PROGRESS.PROGRESS_PREPARE:


    IF (_eRslt = E_PROGRESS.PROGRESS_ERROR)
    THEN
      _eState                   := E_PROGRESS.PROGRESS_ERROR;
      _nErrorId                 := _MoverInfo[_nMover].nErrorId; 

    ELSIF (_eRslt = E_PROGRESS.PROGRESS_DONE)
    THEN
      _eState                   := E_PROGRESS.PROGRESS_STARTUP;
    END_IF
END_CASE
//-----------------------------------------------------------------------------
//-----------------------------------------------------------------------------
CASE _eState
OF
  E_PROGRESS.PROGRESS_STARTUP:
    _eState                     := E_PROGRESS.PROGRESS_CHECK;

END_CASE
//-----------------------------------------------------------------------------
//-----------------------------------------------------------------------------
CASE _eState
OF
  E_PROGRESS.PROGRESS_CHECK:
    IF (_nMover > MAX_MOVER-1)
    THEN
      _eState                   := E_PROGRESS.PROGRESS_DONE;
    ELSE
      _nMover                   := _nMover + 1;
      _eState                   := E_PROGRESS.PROGRESS_BUSY;
    END_IF
END_CASE
//-----------------------------------------------------------------------------
//-----------------------------------------------------------------------------

TransportRestart                := _eState;
END_METHOD

METHOD TransportStart : e_progress
VAR_INPUT
  Execute       : BOOL;
END_VAR
VAR_INST
  _nMover,
  _nStation     : UINT;
  _nErrorId     : UDINT;

  _stMoveData   : ST_MOVE_DATA;

  _eRslt,
  _eState       : E_PROGRESS;

END_VAR
//-----------------------------------------------------------------------------
IF NOT Execute 
THEN 
	_eState                       := E_PROGRESS.PROGRESS_INIT; 
END_IF 
//-----------------------------------------------------------------------------
IF NOT Check() 
THEN 
	TransportStart                := E_PROGRESS.PROGRESS_ERROR; 
	RETURN; 
END_IF
//-----------------------------------------------------------------------------
//-----------------------------------------------------------------------------
CASE _eState
OF
  E_PROGRESS.PROGRESS_INIT:
    IF Execute
    THEN
      _nErrorId                 := 0;
      _nMover                   := 1;

      _stMoveData.rPos          := _StationStart.rPosWait + _MoverItf[_nMover].RailLength;
      _stMoveData.rGap          := _StationStart.rGap;

      _stMoveData.rVelo         := _StationStart.rVelo;
      _stMoveData.rAcc          := _StationStart.rAccDec;
      _stMoveData.rJerk         := _StationStart.rJerk;

      _stMoveData.rDelta        :=   0.05;
      _stMoveData.rDistance     :=  -1.0;     // distance used by SendToPosCa

      _stMoveData.rOverride     := 100.0;

      FOR _nStation := 1 TO MAX_STATION
      DO
        _ItfStationCtrl[_nStation].Init();    // clear all stations
      END_FOR

      _eState                   := E_PROGRESS.PROGRESS_BUSY;
    END_IF

  //---------------------------------------------------------------------------
  E_PROGRESS.PROGRESS_BUSY:
    _eState                     := E_PROGRESS.PROGRESS_PREPARE;
    _eRslt                      := _MoverItf[_nMover].SendToModuloPosCa(FALSE, _stMoveData);
    _eRslt                      := _MoverItf[_nMover].SendToAbsPosCa(FALSE, _stMoveData);

  E_PROGRESS.PROGRESS_PREPARE:
    _eRslt                      := _MoverItf[_nMover].SendToModuloPosCa(TRUE, _stMoveData);

    IF (_eRslt = E_PROGRESS.PROGRESS_ERROR)
    THEN
      _eState                   := E_PROGRESS.PROGRESS_ERROR;
      _nErrorId                 := _MoverInfo[_nMover].nErrorId;
      _eRslt                    := _MoverItf[_nMover].SendToModuloPosCa(FALSE, _stMoveData); 

    ELSIF (_eRslt = E_PROGRESS.PROGRESS_DONE)
    THEN
      _eState                   := E_PROGRESS.PROGRESS_STARTUP;
      _eRslt                    := _MoverItf[_nMover].SendToModuloPosCa(FALSE, _stMoveData);
    END_IF

  //---------------------------------------------------------------------------
  E_PROGRESS.PROGRESS_STARTUP:
    IF (_nMover > MAX_MOVER-1)
    THEN
      // all mover are sent to start position, now prepare ticket for Mover 1
      _eState                         := E_PROGRESS.PROGRESS_CHECK;
      // ticket data
      _stMoverDataSend.nMask          := TO_USINT(EXPT(2,_StationStart.nConfiguredStopCount))-1;
      _stMoverDataSend.nMoverId       := TO_USINT(1);
      _stMoverDataSend.nTargetStation := TO_USINT(_nStartStation);
  
      _stListResult                   := _ItfStationList[_nStartStation].AddTailValue(_stMoverDataSend); // add first mover to list of _ItfStations[_nStartStation]

    ELSE
      _nMover                   := _nMover + 1;                                                 // increment mover ID
      _stMoveData.rPos          := _StationStart.rPosWait + 2*_MoverItf[_nMover].RailLength;    // all other mover are commanded an extra round, to make sure that mover 1 is always leading the pack
      _eState                   := E_PROGRESS.PROGRESS_BUSY;                                    // go back and trigger move
    END_IF

  //---------------------------------------------------------------------------
  E_PROGRESS.PROGRESS_CHECK:
    IF (_MoverInfo[1].rAbsActPos > _MoverInfo[1].rAbsTargetPos - 1.0) AND
       (_MoverInfo[1].rAbsActPos < _MoverInfo[1].rAbsTargetPos + 1.0) // wait for first mover to arrive
    THEN
      IF (_GroupInfo.AllAxesStanding) // wait for all mover standstill
      THEN
        _stMoveData.rPos        := _MoverInfo[1].rAbsTargetPos;                    // Mover1 position to retrigger the movers
        _nMover                 := 2;
        _eState                 := E_PROGRESS.PROGRESS_OCCUPIED;
      END_IF
    END_IF

  //---------------------------------------------------------------------------
  E_PROGRESS.PROGRESS_OCCUPIED:
    _eRslt                      := _MoverItf[_nMover].SendToAbsPosCa(TRUE, _stMoveData); // retrigger

    IF (_eRslt = E_PROGRESS.PROGRESS_ERROR)
    THEN
      _eState                   := E_PROGRESS.PROGRESS_ERROR;
      _nErrorId                 := _MoverInfo[_nMover].nErrorId;
      _eRslt                    := _MoverItf[_nMover].SendToAbsPosCa(FALSE, _stMoveData); 

    ELSIF (_eRslt = E_PROGRESS.PROGRESS_DONE)
    THEN
      _eState                   := E_PROGRESS.PROGRESS_WORKING;
      _eRslt                    := _MoverItf[_nMover].SendToAbsPosCa(FALSE, _stMoveData);

      // write ticket for mover in station list
      _stMoverDataSend.nMask          := TO_USINT(EXPT(2,_StationStart.nConfiguredStopCount))-1;
      _stMoverDataSend.nMoverId       := TO_USINT(_nMover);
      _stMoverDataSend.nTargetStation := TO_USINT(_nStartStation);
  
      _stListResult                   := _ItfStationList[_nStartStation].AddTailValue(_stMoverDataSend); // enter in list
    END_IF

  //---------------------------------------------------------------------------
  E_PROGRESS.PROGRESS_WORKING:
    IF (_nMover > MAX_MOVER-1)
    THEN
      _eState                   := E_PROGRESS.PROGRESS_DONE;
    ELSE
      _nMover                   := _nMover + 1;
      _eState                   := E_PROGRESS.PROGRESS_OCCUPIED;
    END_IF
END_CASE
//-----------------------------------------------------------------------------
//-----------------------------------------------------------------------------

TransportStart                  := _eState;
END_METHOD

PROPERTY XpuCtrl : REFERENCE TO ST_XPU_CTRL
SET
_XpuCtrl REF= XpuCtrl;
END_SET
END_PROPERTY

PROPERTY XpuInfo : REFERENCE TO ST_XPU_INFO
SET
_XpuInfo REF= XpuInfo;
END_SET
END_PROPERTY

METHOD XpuInit : E_PROGRESS
VAR_INPUT
  Execute     : BOOL;
END_VAR
VAR_INST
  _nErrorId   : UDINT;
  _eJobReslt,
  _eState     : E_PROGRESS;
END_VAR
//-----------------------------------------------------------------------------
IF NOT Execute 
THEN 
	_eState                       := E_PROGRESS.PROGRESS_INIT; 
END_IF 
//-----------------------------------------------------------------------------
IF NOT Check() 
THEN 
	XpuInit                       := E_PROGRESS.PROGRESS_ERROR; 
	RETURN; 
END_IF
//-----------------------------------------------------------------------------
//-----------------------------------------------------------------------------
CASE _eState
OF
  E_PROGRESS.PROGRESS_INIT:
    IF Execute
    THEN
      _nErrorId                 := 0;
      _XpuCtrl.Cmd              := E_XPU_CTRL.XTS_CMD_NULL; // clear interface

      _eState                   := E_PROGRESS.PROGRESS_BUSY;
    END_IF
  //---------------------------------------------------------------------------
  //---------------------------------------------------------------------------
  E_PROGRESS.PROGRESS_BUSY:
    _XpuCtrl.Cmd                := E_XPU_CTRL.XTS_CMD_INIT; // start Xpu init

    IF (f_GetProgress(_XpuState.State) = E_PROGRESS.PROGRESS_DONE)         // check Xpu init done
    THEN
      _eState                   := E_PROGRESS.PROGRESS_PREPARE;

    ELSIF (f_GetProgress(_XpuState.State) = E_PROGRESS.PROGRESS_ERROR)     // check for error
    THEN
      _eState                   := E_PROGRESS.PROGRESS_ERROR;
    END_IF
  //---------------------------------------------------------------------------
  //---------------------------------------------------------------------------
  E_PROGRESS.PROGRESS_PREPARE:
    _XpuCtrl.Cmd                := E_XPU_CTRL.XTS_IDLE;     // Xpu start cyclic checks and mover detection

    IF (f_GetProgress(_XpuState.State) = E_PROGRESS.PROGRESS_ERROR)     // check for error
    THEN
      _eState                   := E_PROGRESS.PROGRESS_ERROR;

    ELSIF (f_GetProgress(_XpuState.State) = E_PROGRESS.PROGRESS_WORKING)      // check Xpu Idle working
    THEN
      _eState                   := E_PROGRESS.PROGRESS_STARTUP;

    END_IF
  //---------------------------------------------------------------------------
  //---------------------------------------------------------------------------
  E_PROGRESS.PROGRESS_STARTUP:
    IF (f_GetProgress(_XpuState.State) = E_PROGRESS.PROGRESS_ERROR)
    THEN
      _eState                   := E_PROGRESS.PROGRESS_ERROR;

    ELSIF (_XpuState.Check = E_XPU_CHECK.MOVER_ID_SIMULATION) OR
          (_XpuState.Check = E_XPU_CHECK.MOVER_ID_STANDARD)   OR
          (_XpuState.Check = E_XPU_CHECK.MOVER_ID_DETECTION_VALID)
    THEN
      _eState                   := E_PROGRESS.PROGRESS_DONE;
    END_IF
END_CASE
//-----------------------------------------------------------------------------
//-----------------------------------------------------------------------------
XpuInit                         := _eState;
END_METHOD

PROPERTY XpuState : REFERENCE TO ST_XPU_STATE
SET
_XpuState ref= XpuState;
END_SET
END_PROPERTY

END_FUNCTION_BLOCK

